    |     # get second point (right) (point2)
    |     # take the center point and move right the radius plus the cushions
    |     p2x = pcx + vecrx * radius + vecrx * cusharound + vecnx * -1 * cushout
    |     p2y = pcy + vecry * radius + vecry * cusharound + vecny * -1 * cushout
    |     p2z = pcz
    | 
    |     # find rxryrz2
    |     # first rotation is 90 degrees about the x- axis
    |     m1 = get_rotation_matrix_from_description("x", -1, 90 * pi / 180)
    |     # second rotation is About 135 degrees about the z+ axis. This calculation is heading1 – 45 degrees
    |     m2 = get_rotation_matrix_from_description("z", 1, heading1 - 45 * pi/180)
    |     # combine them by multiplying
    |     m3 = multiply_matrix(m2, m1)
    |     rxryrz2 = convert_matrix_to_axang(m3)
    |     rx2 = rxryrz2[0]
    |     ry2 = rxryrz2[1]
    |     rz2 = rxryrz2[2]
    | 
    |     point2 = p[p2x, p2y, p2z, rx2, ry2, rz2]
    | 
    |     # get the third point (bottom) (point3)
    |     p3x = pcx + vecnx * -1 * cushout
    |     p3y = pcy + vecny * -1 * cushout
    |     p3z = pcz - vecuz * radius - vecuz * cusharound
    | 
    |     # find rxryrz3
    |     # first rotation is 45 degrees about the y+ axis
    |     m1 = get_rotation_matrix_from_description("y", 1, 45 * pi / 180)
    |     # second rotation is About 180 degrees about the z+ axis. This calculation is heading1 degrees
    |     m2 = get_rotation_matrix_from_description("z", 1, heading1)
    |     # combine them by multiplying
    |     m3 = multiply_matrix(m2, m1)
    |     rxryrz3 = convert_matrix_to_axang(m3)
    |     rx3 = rxryrz3[0]
    |     ry3 = rxryrz3[1]
    |     rz3 = rxryrz3[2]
    | 
    |     point3 = p[p3x, p3y, p3z, rx3, ry3, rz3]
    | 
    |     # get the fourth point (left) (point4)
    |     p4x = pcx - vecrx * radius - vecrx * cusharound + vecnx * -1 * cushout
    |     p4y = pcy - vecry * radius - vecry * cusharound + vecny * -1 * cushout
    |     p4z = pcz
    | 
    |     # find rxryrz4
    |     # first rotation is 90 degrees about the x+ axis
    |     m1 = get_rotation_matrix_from_description("x", 1, 90 * pi / 180)
    |     # second rotation is heading1 + 45 degrees about the z+ axis. approx 225 degrees ccw
    |     m2 = get_rotation_matrix_from_description("z", 1, heading1 + 45 * pi/180)
    |     # combine them by multiplying
    |     m3 = multiply_matrix(m2, m1)
    |     rxryrz4 = convert_matrix_to_axang(m3)
    |     rx4 = rxryrz4[0]
    |     ry4 = rxryrz4[1]
    |     rz4 = rxryrz4[2]
    | 
    |     point4 = p[p4x, p4y, p4z, rx4, ry4, rz4]
    | 
    |     # return the points
    |     ret = struct(point1=point1, point2=point2, point3=point3, point4=point4)
    |     return ret
    | 
    | end
  SuppressedNode
    Script: welder_state_ready()
  SuppressedNode
    sidewallchoice :=  (valueSource=Operator message=Is the sidewall 3/4 inch? valueType=Boolean)
  SuppressedNode
    If sidewallchoice removedSiblings(If(type=Else checkContinuously=false, children(Assignment(valueSource=Expression, variable(name=sidewall), expression=0.375))))
      sidewall := 0.628
  SuppressedNode
    deepcham :=  (valueSource=Operator message=Is the chamfer extra deep? (more than 0.21) valueType=Boolean)
  MoveJ speed 60 deg/s, acceleration 80 deg/s^2 (useActiveTCP=true optimoveEnabled=false optiMoveSpeed=0.3 optiMoveAcceleration=0.09) feature=Base
    Waypoint Waypoint_46: TCP in base x=894.108 y=351.078 z=354.456 mm, rx=2.3264 ry=2.0525 rz=0.0574 rad; joints [-187.182, -67.294, 94.726, 57.522, -0.141, -88.018] deg; TCP offset x=-5.49 y=-328 z=106.39 mm, rx=1.2092 ry=-1.2092 rz=1.2092 rad
  Set NoAction tcp=pretend_w_top
  Script: Test_Teach_Sleeve_Fillet()
  Set NoAction tcp=pretend_w_top
  Script: kill threadId_Thread_1
  Set NoAction tcp=pretend_welder
  SuppressedNode
    path1 := analyze_touchpoints(p11,p12,p21,p22,p3)
  SuppressedNode
    CallSubProgram
  SuppressedNode
    MoveJ speed 60 deg/s, acceleration 80 deg/s^2 (useActiveTCP=true optimoveEnabled=false optiMoveSpeed=0.3 optiMoveAcceleration=0.09) feature=Base
      Waypoint Waypoint_19: TCP in base x=-539.433 y=254.004 z=21.521 mm, rx=-1.7232 ry=0.9213 rz=1.7071 rad; joints [-41.97, -63.602, 146.502, 9.159, 84.533, 189.272] deg; TCP offset x=8.55 y=-271.52 z=102 mm, rx=1.2092 ry=-1.2092 rz=1.2092 rad
  pathturn := main_calculate_sleeve_fillet(tcp_pose_left, tcp_pose_right, tcp_3)
  SuppressedNode
    Folder extrude knife
      lch := get_lift_column_height_condensed()
      If lch > 1
        URCap MachineLogic for Universal Robots (MachineLogic for Universal Robots, Vention Inc.) dataModel(type=addMotor, numberAdded=0, speed_in_mm_per_min=3000.0, acceleration_in_mm_per_s2=50.0, teachColor=BLUE, combo1=MachineMotion1, combo2=(1) Custom Actuator, combo3=Home, combo6=In series, message=Homing, description=Moves the actuator in the negative direction until the home sensor is triggered and sets position to zero (0)., comboAddress=Address 1, comboActuator=Valve 1)
        Script: extrude_knife3()
        URCap MachineLogic for Universal Robots (MachineLogic for Universal Robots, Vention Inc.) dataModel(type=addMotor, numberAdded=0, speed_in_mm_per_min=3000.0, acceleration_in_mm_per_s2=50.0, ActuatorPos=lch, teachColor=BLUE, combo1=MachineMotion1, combo2=(1) Custom Actuator, combo3=Move to Position, combo6=In series, message=Move to Position, description=Moves the actuator to a specified position from the home location., comboAddress=Address 1, comboActuator=Valve 1)
      Else 
        Script: extrude_knife3()
  Script: extrude_knife3()
  SuppressedNode
    Script: move_path_cover_left3()
  SuppressedNode
    pointtopvcham := pathturn[0]
  SuppressedNode
    URCap MachineLogic for Universal Robots (MachineLogic for Universal Robots, Vention Inc.) dataModel(type=addMotor, numberAdded=0, speed_in_mm_per_min=3000.0, acceleration_in_mm_per_s2=50.0, ActuatorPos=liftcolumnzneeded, teachColor=BLUE, combo1=MachineMotion1, combo2=(1) Custom Actuator, combo3=Move to Position, combo6=In series, message=Move to Position, description=Moves the actuator to a specified position from the home location., comboAddress=Address 1, comboActuator=Valve 1)
  SuppressedNode
    MoveJ speed 60 deg/s, acceleration 80 deg/s^2 (useActiveTCP=true optimoveEnabled=false optiMoveSpeed=0.3 optiMoveAcceleration=0.09) feature=Base
      Waypoint Variable (Variable): variable=pointtopvcham
  Script: align_sleeve_fillet_low()
  Script: move_sleeve_fillet_quad()
  MoveJ speed 60 deg/s, acceleration 80 deg/s^2 (useActiveTCP=true optimoveEnabled=false optiMoveSpeed=0.3 optiMoveAcceleration=0.09) feature=Base
    Waypoint Waypoint_8: TCP in base x=-262.599 y=-117.911 z=443.767 mm, rx=0.1153 ry=3.1146 rz=0.2657 rad; joints [5.497, -142.032, 129.309, 13.11, 99.793, -9.621] deg; TCP offset x=-9.5 y=-328 z=105.73 mm, rx=1.2092 ry=-1.2092 rz=1.2092 rad
    Waypoint Waypoint_9: TCP in base x=397.354 y=356.263 z=319.809 mm, rx=2.3163 ry=2.0576 rz=0.0741 rad; joints [-198.308, -118.162, 133.452, -12.561, -11.517, -6.326] deg
  SuppressedNode
    URCap MachineLogic for Universal Robots (MachineLogic for Universal Robots, Vention Inc.) dataModel(type=addMotor, numberAdded=0, speed_in_mm_per_min=3000.0, acceleration_in_mm_per_s2=50.0, teachColor=BLUE, combo1=MachineMotion1, combo2=(1) Custom Actuator, combo3=Home, combo6=In series, message=Homing, description=Moves the actuator in the negative direction until the home sensor is triggered and sets position to zero (0)., comboAddress=Address 1, comboActuator=Valve 1)
  SafeHome (positionOptionType=SPEED_AND_ACCELERATION speed=1.047198 acceleration=1.396263 nextMotionTime=2)
SubProgram Test_Teach_Sleeve_Fillet (keepSynchronizedWithDisk=false) programFile=/programs/Test Teach Sleeve Fillet.urp
  Set NoAction tcp=pretend_w_top
  SuppressedNode
    MoveL speed 250 mm/s, acceleration 1200 mm/s^2 (useActiveTCP=true optimoveEnabled=false optiMoveSpeed=0.3 optiMoveAcceleration=0.09) feature=Base
      Waypoint Waypoint_1: TCP in base x=183.613 y=373.491 z=464.002 mm, rx=0 ry=3.1416 rz=0 rad; joints [-144.817, -120.486, 148.461, -117.931, -90.033, 125.101] deg; TCP offset x=0 y=0 z=19 mm, rx=0 ry=0 rz=0 rad
      'move welder up out of holder'
  MoveJ speed 60 deg/s, acceleration 80 deg/s^2 (useActiveTCP=false optimoveEnabled=false optiMoveSpeed=0.3 optiMoveAcceleration=0.09) tcp=TCP_1_plate; feature=Base
    Waypoint Waypoint_40: TCP in base x=360.688 y=270.12 z=646.145 mm, rx=0.0578 ry=2.126 rz=2.1341 rad; joints [-198.126, -117.852, 133.303, -13.01, -11.422, -6.036] deg
    'above waypoint is home'
    SuppressedNode
      Waypoint Waypoint_2: TCP in base x=-548.957 y=386.285 z=143.71 mm, rx=1.5708 ry=0 rz=0 rad; joints [-60.253, -57.926, 123.544, -65.529, -60.311, -0.099] deg
    SuppressedNode
      Waypoint Waypoint_3: TCP in base x=-565.561 y=-88.282 z=748.934 mm, rx=0.347 ry=3.1015 rz=-0.0385 rad; joints [-12.028, -113.359, 121.362, 263.351, -88.693, -89.284] deg
    Waypoint Waypoint_4: TCP in base x=-946.63 y=32.923 z=107.553 mm, rx=1.1855 ry=-1.4546 rz=-1.2991 rad; joints [-14.723, -32.384, 121.91, 97.274, -87.344, -180.783] deg
  Set NoAction tcp=pretend_w_top
  freedrive_m_var := False
  freedrive_m_var := True
  Popup Message (haltProgram=false message=Move the TCP to point 1 on the edge then click 'Continue' inputType=Text)
  tcp_pose_left := get_actual_tcp_pose()
  freedrive_m_var := False
  Script: sync()
  Wait Sleep waitTime=0.01
  MoveJ speed 60 deg/s, acceleration 80 deg/s^2 (useActiveTCP=true optimoveEnabled=false optiMoveSpeed=0.3 optiMoveAcceleration=0.09) feature=Base
    Waypoint Waypoint_4: TCP in base x=-946.63 y=32.923 z=107.553 mm, rx=1.1855 ry=-1.4546 rz=-1.2991 rad; joints [-14.723, -32.384, 121.91, 97.274, -87.344, -180.783] deg
  MoveJ speed 60 deg/s, acceleration 80 deg/s^2 (useActiveTCP=true optimoveEnabled=false optiMoveSpeed=0.3 optiMoveAcceleration=0.09) feature=Base
    Waypoint Waypoint_5: TCP in base x=-1246.557 y=36.36 z=-286.524 mm, rx=0.3629 ry=-1.2595 rz=-1.7222 rad; joints [1.222, -11.211, 100.501, 238.355, -233.303, -3.079] deg; TCP offset x=-1.032 y=-18.062 z=285.234 mm, rx=0 ry=0 rz=0 rad
  freedrive_m_var := True
  Popup Message (haltProgram=false message=Move the TCP to point 2 on the edge then click 'Continue' inputType=Text)
  tcp_pose_right := get_actual_tcp_pose()
  Popup Message (haltProgram=false message=Move the TCP to point 3 on the edge then click 'Continue' inputType=Text)
  tcp_3 := get_actual_tcp_pose()
  freedrive_m_var := False
  Wait Sleep waitTime=0.25
  Script: sync()
  MoveL speed 100 mm/s, acceleration 1200 mm/s^2 (useActiveTCP=true optimoveEnabled=false optiMoveSpeed=0.3 optiMoveAcceleration=0.09) feature=Base
    MoveDirectionNode expression=[1.0,0.0,-0.5]
      Until DISTANCE (allowActions=false deceleration=3 distanceNodeType=STOP) Distance=0.15; motionParameters(blendRadius=0)
  MoveJ speed 60 deg/s, acceleration 80 deg/s^2 (useActiveTCP=true optimoveEnabled=false optiMoveSpeed=0.3 optiMoveAcceleration=0.09) feature=Base
    Waypoint Waypoint_5: TCP in base x=-1246.557 y=36.36 z=-286.524 mm, rx=0.3629 ry=-1.2595 rz=-1.7222 rad; joints [1.222, -11.211, 100.501, 238.355, -233.303, -3.079] deg
    Waypoint Waypoint_4: TCP in base x=-946.63 y=32.923 z=107.553 mm, rx=1.1855 ry=-1.4546 rz=-1.2991 rad; joints [-14.723, -32.384, 121.91, 97.274, -87.344, -180.783] deg; TCP offset x=0 y=0 z=19 mm, rx=0 ry=0 rz=0 rad
    Waypoint Waypoint_1: TCP in base x=394.188 y=534.376 z=630.191 mm, rx=0.0578 ry=2.126 rz=2.1341 rad; joints [-198.279, -117.801, 133.277, -12.745, -11.485, -6.332] deg; TCP offset x=-1.032 y=-18.062 z=285.234 mm, rx=0 ry=0 rz=0 rad
SubProgram move_sleeve_fillet_quad (keepSynchronizedWithDisk=false) programFile=/programs/move_sleeve_fillet_quad.urp
  Set NoAction tcp=backofhole
  SuppressedNode
    MoveJ speed 60 deg/s, acceleration 80 deg/s^2 (useActiveTCP=true optimoveEnabled=false optiMoveSpeed=0.3 optiMoveAcceleration=0.09) feature=Base
      SuppressedNode
        Waypoint Waypoint_3: TCP in base x=-912.453 y=673.518 z=718.985 mm, rx=-0.4706 ry=-1.9428 rz=0.4955 rad; joints [-63.285, -68.284, 110.161, 88.985, -83.541, -118.353] deg; TCP offset x=-9.5 y=-328 z=105.73 mm, rx=1.2092 ry=-1.2092 rz=1.2092 rad
      SuppressedNode
        Waypoint Waypoint_4: TCP in base x=-1043.534 y=752.126 z=758.241 mm, rx=-0.4498 ry=-2.3257 rz=-0.2665 rad; joints [-53.991, -67.414, 94.218, 102.936, -66.691, -159.337] deg
      Waypoint Waypoint_9: TCP in base x=-850.146 y=808.476 z=769.845 mm, rx=-0.0694 ry=-2.4231 rz=-0.6317 rad; joints [-70.02, -72.001, 93.194, -274.04, -37.901, -142.904] deg
      Waypoint Waypoint_6: TCP in base x=-1042.273 y=808.476 z=769.845 mm, rx=-0.0694 ry=-2.4231 rz=-0.6317 rad; joints [-58.413, -64.349, 84.656, -260.501, -42.539, -159.423] deg
  SuppressedNode
    MoveJ speed 60 deg/s, acceleration 80 deg/s^2 (useActiveTCP=true optimoveEnabled=false optiMoveSpeed=0.3 optiMoveAcceleration=0.09) feature=Base
      SuppressedNode
        Waypoint Waypoint_1: TCP in base x=-1152.594 y=814.679 z=699.964 mm, rx=0.098 ry=-2.3843 rz=-0.4483 rad; joints [-56.525, -54.403, 73.307, 93.455, -42.841, -145.624] deg
      SuppressedNode
        Waypoint Waypoint_5: TCP in base x=-1149.758 y=814.958 z=702.794 mm, rx=-0.0472 ry=-2.3472 rz=-0.7271 rad; joints [-53.278, -57.004, 80.845, -264.711, -44.526, -166.31] deg
      Waypoint Waypoint_7: TCP in base x=-1150.142 y=824.468 z=703.476 mm, rx=-0.1355 ry=-2.1954 rz=-0.513 rad; joints [-54.373, -54.473, 80.141, -274.253, -56.089, -154.835] deg
  SuppressedNode
    MoveP speed 10 mm/s, acceleration 1200 mm/s^2 (blendRadius=0.025 useActiveTCP=true optimoveEnabled=false optiMoveSpeed=0.3 optiMoveAcceleration=0.09) feature=Base
      CircleMove (OrientationMode=FIXED)
        Waypoint ViaPoint_1: TCP in base x=-1137.967 y=888.777 z=671.431 mm, rx=-0.7156 ry=-2.1833 rz=0.6859 rad; joints [-57.632, -55.198, 82.444, 124.608, -82.298, -128.207] deg
        Waypoint EndPoint_1: TCP in base x=-1139.924 y=872.884 z=596.072 mm, rx=-1.219 ry=-0.9297 rz=2.3215 rad; joints [-60.159, -58.197, 98.87, 176.452, -78.393, -68.042] deg
      CircleMove (OrientationMode=FIXED)
        Waypoint ViaPoint_2: TCP in base x=-1155.211 y=763.52 z=646.144 mm, rx=0.9307 ry=-1.6945 rz=-2.1414 rad; joints [-52.747, -75.971, 108.96, 234.472, -18.82, -4.377] deg
        Waypoint Waypoint_1: TCP in base x=-1152.594 y=814.679 z=699.964 mm, rx=0.098 ry=-2.3843 rz=-0.4483 rad; joints [-56.525, -54.403, 73.307, 93.455, -42.841, -145.624] deg
  SuppressedNode
    MoveJ speed 60 deg/s, acceleration 80 deg/s^2 (useActiveTCP=true optimoveEnabled=false optiMoveSpeed=0.3 optiMoveAcceleration=0.09) feature=Base
      SuppressedNode
        Waypoint Waypoint_2: TCP in base x=-917.75 y=830.261 z=524.512 mm, rx=-1.543 ry=-0.8444 rz=1.9881 rad; joints [-66.08, -72.484, 118.808, 175.962, -93.351, -73.55] deg
      Waypoint Waypoint_4: TCP in base x=-1043.534 y=752.126 z=758.241 mm, rx=-0.4498 ry=-2.3257 rz=-0.2665 rad; joints [-53.991, -67.414, 94.218, 102.936, -66.691, -159.337] deg
      Waypoint Waypoint_8: TCP in base x=-754.583 y=757.082 z=772.781 mm, rx=-0.4498 ry=-2.3257 rz=-0.2665 rad; joints [-73.782, -79.343, 107.572, 92.439, -55.198, -140.846] deg
  SuppressedNode
    Folder half circle
      MoveJ speed 60 deg/s, acceleration 80 deg/s^2 (useActiveTCP=true optimoveEnabled=false optiMoveSpeed=0.3 optiMoveAcceleration=0.09) feature=Base
        Waypoint Waypoint_13: TCP in base x=-1410.884 y=263.861 z=-13.194 mm, rx=-0.2057 ry=-2.2742 rz=-0.4378 rad; joints [-18.611, -21.126, 85.064, -293.08, -78.09, -188.172] deg
      MoveJ speed 60 deg/s, acceleration 80 deg/s^2 (useActiveTCP=true optimoveEnabled=false optiMoveSpeed=0.3 optiMoveAcceleration=0.09) feature=Base
        Waypoint Waypoint_10: TCP in base x=-1440.647 y=263.861 z=-48.062 mm, rx=-0.2057 ry=-2.2742 rz=-0.4378 rad; joints [-18.086, -18.126, 80.761, -291.695, -78.433, -188.577] deg
        SuppressedNode
          Waypoint Waypoint_11: TCP in base x=-1286.175 y=549.195 z=115.468 mm, rx=-0.27 ry=-1.5277 rz=-1.42 rad; joints [-20.499, -22.138, 88.563, -259.74, -128.557, -138.212] deg; TCP offset x=-1.032 y=-18.062 z=285.234 mm, rx=0 ry=0 rz=0 rad
        SuppressedNode
          Waypoint Waypoint_12: TCP in base x=-1198.19 y=495.746 z=-342.486 mm, rx=-1.4417 ry=-1.7142 rz=-0.5215 rad; joints [-20.358, -19.189, 100.698, -215.464, -126.338, -45.331] deg
      MoveP speed 8 mm/s, acceleration 1200 mm/s^2 (blendRadius=0.025 useActiveTCP=true optimoveEnabled=false optiMoveSpeed=0.3 optiMoveAcceleration=0.09) feature=Base
        CircleMove (OrientationMode=FIXED)
          Waypoint ViaPoint_3: TCP in base x=-1436.982 y=288.423 z=-164.849 mm, rx=-1.2985 ry=-1.3493 rz=1.8084 rad; joints [-22.4, -18.108, 96.782, -229.781, -128.579, -68.735] deg; TCP offset x=-9.5 y=-328 z=105.73 mm, rx=1.2092 ry=-1.2092 rz=1.2092 rad
          Waypoint EndPoint_2: TCP in base x=-1450.471 y=225.502 z=-193.907 mm, rx=-1.3296 ry=-0.3697 rz=2.6077 rad; joints [-22.267, -13.945, 97.987, -213.988, -92.35, -25.678] deg
      MoveJ speed 60 deg/s, acceleration 80 deg/s^2 (useActiveTCP=true optimoveEnabled=false optiMoveSpeed=0.3 optiMoveAcceleration=0.09) feature=Base
        Waypoint Waypoint_14: TCP in base x=-1380.88 y=218.821 z=-252.804 mm, rx=-1.3435 ry=-0.3935 rz=2.6113 rad; joints [-23.838, -10.524, 100.952, -220.078, -91.217, -28.02] deg
  Folder assign points
    p1 := pathturn[0]
    p2 := pathturn[1]
    p3 := pathturn[2]
    p4 := pathturn[3]
    pa1 := p[p1[0]+0.05,p1[1],p1[2]+0.05,p1[3],p1[4],p1[5]]
  Folder full circle
    SuppressedNode
      MoveJ speed 60 deg/s, acceleration 80 deg/s^2 (useActiveTCP=true optimoveEnabled=false optiMoveSpeed=0.3 optiMoveAcceleration=0.09) feature=Base
        'start point example'
        Waypoint Waypoint_13: TCP in base x=-1410.884 y=263.861 z=-13.194 mm, rx=-0.2057 ry=-2.2742 rz=-0.4378 rad; joints [-18.611, -21.126, 85.064, -293.08, -78.09, -188.172] deg
    MoveJ speed 60 deg/s, acceleration 80 deg/s^2 (useActiveTCP=true optimoveEnabled=false optiMoveSpeed=0.3 optiMoveAcceleration=0.09) feature=Base
      SuppressedNode
        Waypoint Waypoint_10: TCP in base x=-1440.647 y=263.861 z=-48.062 mm, rx=-0.2057 ry=-2.2742 rz=-0.4378 rad; joints [-18.086, -18.126, 80.761, -291.695, -78.433, -188.577] deg
      SuppressedNode
        Waypoint Waypoint_11: TCP in base x=-1286.175 y=549.195 z=115.468 mm, rx=-0.27 ry=-1.5277 rz=-1.42 rad; joints [-20.499, -22.138, 88.563, -259.74, -128.557, -138.212] deg; TCP offset x=-1.032 y=-18.062 z=285.234 mm, rx=0 ry=0 rz=0 rad
      SuppressedNode
        Waypoint Waypoint_12: TCP in base x=-1198.19 y=495.746 z=-342.486 mm, rx=-1.4417 ry=-1.7142 rz=-0.5215 rad; joints [-20.358, -19.189, 100.698, -215.464, -126.338, -45.331] deg
      Waypoint Variable (Variable): variable=pa1
      Waypoint Variable (Variable): variable=p1
    SuppressedNode
      MoveP speed 8 mm/s, acceleration 1200 mm/s^2 (blendRadius=0.025 useActiveTCP=true optimoveEnabled=false optiMoveSpeed=0.3 optiMoveAcceleration=0.09) feature=Base
        CircleMove (OrientationMode=FIXED)
          Waypoint ViaPoint_3: TCP in base x=-1436.982 y=288.423 z=-164.849 mm, rx=-1.2985 ry=-1.3493 rz=1.8084 rad; joints [-22.4, -18.108, 96.782, -229.781, -128.579, -68.735] deg; TCP offset x=-9.5 y=-328 z=105.73 mm, rx=1.2092 ry=-1.2092 rz=1.2092 rad
          Waypoint EndPoint_2: TCP in base x=-1450.471 y=225.502 z=-193.907 mm, rx=-1.3296 ry=-0.3697 rz=2.6077 rad; joints [-22.267, -13.945, 97.987, -213.988, -92.35, -25.678] deg
        CircleMove (OrientationMode=FIXED)
          Waypoint ViaPoint_4: TCP in base x=-1458.06 y=174.729 z=-155.961 mm, rx=0.9854 ry=-0.8297 rz=-2.4175 rad; joints [-21.89, -10.796, 94.59, -213.949, -40.159, 6.455] deg
          Waypoint EndPoint_3: TCP in base x=-1453.174 y=244.554 z=-53.456 mm, rx=-0.0081 ry=-2.2253 rz=-0.4366 rad; joints [-20.236, -35.116, 108.931, -127.571, 69.187, -2.082] deg
    MoveP speed 10 mm/s, acceleration 1200 mm/s^2 (blendRadius=0.025 useActiveTCP=true optimoveEnabled=false optiMoveSpeed=0.3 optiMoveAcceleration=0.09) feature=Base
      CircleMove (OrientationMode=FIXED)
        Waypoint Variable (Variable): variable=p2
        Waypoint Variable (Variable): variable=p3
      CircleMove (OrientationMode=FIXED)
        Waypoint Variable (Variable): variable=p4
        Waypoint Variable (Variable): variable=p1
    MoveL speed 250 mm/s, acceleration 1200 mm/s^2 (useActiveTCP=true optimoveEnabled=false optiMoveSpeed=0.3 optiMoveAcceleration=0.09) feature=Base
      MoveDirectionNode expression=[1.0,0.0,1.0]
        Until DISTANCE (allowActions=false deceleration=3 distanceNodeType=STOP) Distance=0.1; motionParameters(blendRadius=0)
    Popup Message (haltProgram=true message=pause inputType=Text)
    MoveJ speed 60 deg/s, acceleration 80 deg/s^2 (useActiveTCP=true optimoveEnabled=false optiMoveSpeed=0.3 optiMoveAcceleration=0.09) feature=Base
      Waypoint Waypoint_3: TCP in base x=-1407.381 y=244.554 z=7.478 mm, rx=-0.0081 ry=-2.2253 rz=-0.4366 rad; joints [-21.148, -40.183, 113.996, -127.853, 68.651, -1.292] deg
      Waypoint Waypoint_6: TCP in base x=-1318.966 y=244.554 z=7.478 mm, rx=1.059 ry=-2.1109 rz=-0.921 rad; joints [-32.341, -42.763, 117.442, -171.905, 11.465, 43.721] deg
  SuppressedNode
    MoveJ speed 60 deg/s, acceleration 80 deg/s^2 (useActiveTCP=true optimoveEnabled=false optiMoveSpeed=0.3 optiMoveAcceleration=0.09) feature=Base
      'oldhome'
      Waypoint Waypoint_17: TCP in base x=397.38 y=356.254 z=319.821 mm, rx=2.3163 ry=2.0576 rz=0.0741 rad; joints [-198.308, -118.162, 133.451, -12.562, -11.515, -6.325] deg
  SuppressedNode
    MoveJ speed 60 deg/s, acceleration 80 deg/s^2 (useActiveTCP=true optimoveEnabled=false optiMoveSpeed=0.3 optiMoveAcceleration=0.09) feature=Base
      Waypoint Waypoint_18: TCP in base x=-108.326 y=728.695 z=730.15 mm, rx=-0.9793 ry=0.0055 rz=2.4246 rad; joints [-134.638, -102.677, 135.598, -114.689, -40.923, -114.839] deg
  SuppressedNode
    MoveJ speed 60 deg/s, acceleration 80 deg/s^2 (useActiveTCP=true optimoveEnabled=false optiMoveSpeed=0.3 optiMoveAcceleration=0.09) feature=Base
      Waypoint Waypoint_19: TCP in base x=-1040.406 y=263.861 z=-13.194 mm, rx=-0.2057 ry=-2.2742 rz=-0.4378 rad; joints [-29.173, -26.842, 118.297, -322.804, -71.321, -179.763] deg
  SuppressedNode
    MoveJ speed 60 deg/s, acceleration 80 deg/s^2 (useActiveTCP=true optimoveEnabled=false optiMoveSpeed=0.3 optiMoveAcceleration=0.09) feature=Base
      'example start'
      Waypoint Waypoint_13: TCP in base x=-1410.884 y=263.861 z=-13.194 mm, rx=-0.2057 ry=-2.2742 rz=-0.4378 rad; joints [-18.611, -21.126, 85.064, -293.08, -78.09, -188.172] deg
SubProgram move_path_cover_lt (keepSynchronizedWithDisk=false) programFile=/programs/move_path_cover_lt.urp
  p1 := pathturn[1]
  p2 := pathturn[2]
  p3 := pathturn[3]
  p4 := pathturn[4]
  p5 := pathturn[5]
  p6 := pathturn[6]
  pa1 := p[p1[0],p1[1],p1[2]+0.05,p1[3],p1[4],p1[5]]
  pret := p[p6[0],p6[1],p6[2]+0.05,p6[3],p6[4],p6[5]]
  'go to preheat'
  Set NoAction tcp=pretend_welder
  MoveJ speed 60 deg/s, acceleration 80 deg/s^2 (useActiveTCP=true optimoveEnabled=false optiMoveSpeed=0.3 optiMoveAcceleration=0.09) feature=Base
    Waypoint Variable (Variable): variable=pa1
  MoveL speed 50 mm/s, acceleration 50 mm/s^2 (useActiveTCP=true optimoveEnabled=false optiMoveSpeed=0.3 optiMoveAcceleration=0.09) feature=Base
    Waypoint Variable (Variable): variable=p1
  Wait Sleep waitTime=4
  URCap WireTank Serial (WireTank Serial, WireTank, LLC) dataModel(NODE_TITLE=Serial Bridge uR1, Command=[252,82,49], QUERY=false, byte_array=true, OUTPUT_ENTRY=Static, Variable(key=OUTPUT_VARIABLE, variable(name=HwResp)))
  Set DigitalOutput pin=digital_out[0]; digitalValue=1
  Wait Sleep waitTime=1
  MoveL speed 9 mm/s, acceleration 1200 mm/s^2 (useActiveTCP=true optimoveEnabled=false optiMoveSpeed=0.3 optiMoveAcceleration=0.09) feature=Base
    Waypoint Variable (Variable): variable=p2
    Waypoint Variable (Variable): variable=p3
    Waypoint Variable (Variable): variable=p4
    Waypoint Variable (Variable): variable=p5
  SuppressedNode
    If deepcham removedSiblings(If(type=Else checkContinuously=false, children(Move(motionType=MoveL speed=0.01 acceleration=1.2 useActiveTCP=true positionType=CartesianPose optimoveEnabled=false optiMoveSpeed=0.3 optiMoveAcceleration=0.09, feature=Base, children(Waypoint(type=Variable name=Variable, variable=p2), Waypoint(type=Variable name=Variable, variable=p3), Waypoint(type=Variable name=Variable, variable=p4), Waypoint(type=Variable name=Variable, variable=p5))))))
      MoveL speed 7 mm/s, acceleration 1200 mm/s^2 (useActiveTCP=true optimoveEnabled=false optiMoveSpeed=0.3 optiMoveAcceleration=0.09) feature=Base
        Waypoint Variable (Variable): variable=p2
        Waypoint Variable (Variable): variable=p3
        Waypoint Variable (Variable): variable=p4
        Waypoint Variable (Variable): variable=p5
  URCap WireTank Serial (WireTank Serial, WireTank, LLC) dataModel(QUERY=false, byte_array=true, NODE_TITLE=Serial Bridge uR0, Command=[252,82,48], OUTPUT_ENTRY=Static, Variable(key=OUTPUT_VARIABLE, variable(name=HwResp)))
  Set DigitalOutput pin=digital_out[0]; digitalValue=0
  MoveL speed 10 mm/s, acceleration 1200 mm/s^2 (useActiveTCP=true optimoveEnabled=false optiMoveSpeed=0.3 optiMoveAcceleration=0.09) feature=Base
    Waypoint Variable (Variable): variable=p6
  Wait Sleep waitTime=1
  MoveL speed 50 mm/s, acceleration 50 mm/s^2 (useActiveTCP=true optimoveEnabled=false optiMoveSpeed=0.3 optiMoveAcceleration=0.09) feature=Base
    Waypoint Variable (Variable): variable=pret
SubProgram align_sleeve_fillet_low (keepSynchronizedWithDisk=false) programFile=/programs/align_sleeve_fillet_low.urp
  Set NoAction tcp=pretend_welder
  SuppressedNode
    MoveJ speed 60 deg/s, acceleration 80 deg/s^2 (useActiveTCP=true optimoveEnabled=false optiMoveSpeed=0.3 optiMoveAcceleration=0.09) feature=Base
      SuppressedNode
        Waypoint Waypoint_3: TCP in base x=-912.453 y=673.518 z=718.985 mm, rx=-0.4706 ry=-1.9428 rz=0.4955 rad; joints [-63.285, -68.284, 110.161, 88.985, -83.541, -118.353] deg
      SuppressedNode
        Waypoint Waypoint_4: TCP in base x=-1043.534 y=752.126 z=758.241 mm, rx=-0.4498 ry=-2.3257 rz=-0.2665 rad; joints [-53.991, -67.414, 94.218, 102.936, -66.691, -159.337] deg
      Waypoint Waypoint_9: TCP in base x=-850.146 y=808.476 z=769.845 mm, rx=-0.0694 ry=-2.4231 rz=-0.6317 rad; joints [-70.02, -72.001, 93.194, -274.04, -37.901, -142.904] deg
      Waypoint Waypoint_6: TCP in base x=-1042.273 y=808.476 z=769.845 mm, rx=-0.0694 ry=-2.4231 rz=-0.6317 rad; joints [-58.413, -64.349, 84.656, -260.501, -42.539, -159.423] deg
  SuppressedNode
    MoveJ speed 60 deg/s, acceleration 80 deg/s^2 (useActiveTCP=true optimoveEnabled=false optiMoveSpeed=0.3 optiMoveAcceleration=0.09) feature=Base
      SuppressedNode
        Waypoint Waypoint_1: TCP in base x=-1152.594 y=814.679 z=699.964 mm, rx=0.098 ry=-2.3843 rz=-0.4483 rad; joints [-56.525, -54.403, 73.307, 93.455, -42.841, -145.624] deg
      SuppressedNode
        Waypoint Waypoint_5: TCP in base x=-1149.758 y=814.958 z=702.794 mm, rx=-0.0472 ry=-2.3472 rz=-0.7271 rad; joints [-53.278, -57.004, 80.845, -264.711, -44.526, -166.31] deg
      Waypoint Waypoint_7: TCP in base x=-1150.142 y=824.468 z=703.476 mm, rx=-0.1355 ry=-2.1954 rz=-0.513 rad; joints [-54.373, -54.473, 80.141, -274.253, -56.089, -154.835] deg
  SuppressedNode
    MoveP speed 10 mm/s, acceleration 1200 mm/s^2 (blendRadius=0.025 useActiveTCP=true optimoveEnabled=false optiMoveSpeed=0.3 optiMoveAcceleration=0.09) feature=Base
      CircleMove (OrientationMode=FIXED)
        Waypoint ViaPoint_1: TCP in base x=-1137.967 y=888.777 z=671.431 mm, rx=-0.7156 ry=-2.1833 rz=0.6859 rad; joints [-57.632, -55.198, 82.444, 124.608, -82.298, -128.207] deg
        Waypoint EndPoint_1: TCP in base x=-1139.924 y=872.884 z=596.072 mm, rx=-1.219 ry=-0.9297 rz=2.3215 rad; joints [-60.159, -58.197, 98.87, 176.452, -78.393, -68.042] deg
      CircleMove (OrientationMode=FIXED)
        Waypoint ViaPoint_2: TCP in base x=-1155.211 y=763.52 z=646.144 mm, rx=0.9307 ry=-1.6945 rz=-2.1414 rad; joints [-52.747, -75.971, 108.96, 234.472, -18.82, -4.377] deg
        Waypoint Waypoint_1: TCP in base x=-1152.594 y=814.679 z=699.964 mm, rx=0.098 ry=-2.3843 rz=-0.4483 rad; joints [-56.525, -54.403, 73.307, 93.455, -42.841, -145.624] deg
  SuppressedNode
    MoveJ speed 60 deg/s, acceleration 80 deg/s^2 (useActiveTCP=true optimoveEnabled=false optiMoveSpeed=0.3 optiMoveAcceleration=0.09) feature=Base
      SuppressedNode
        Waypoint Waypoint_2: TCP in base x=-917.75 y=830.261 z=524.512 mm, rx=-1.543 ry=-0.8444 rz=1.9881 rad; joints [-66.08, -72.484, 118.808, 175.962, -93.351, -73.55] deg
      Waypoint Waypoint_4: TCP in base x=-1043.534 y=752.126 z=758.241 mm, rx=-0.4498 ry=-2.3257 rz=-0.2665 rad; joints [-53.991, -67.414, 94.218, 102.936, -66.691, -159.337] deg
      Waypoint Waypoint_8: TCP in base x=-754.583 y=757.082 z=772.781 mm, rx=-0.4498 ry=-2.3257 rz=-0.2665 rad; joints [-73.782, -79.343, 107.572, 92.439, -55.198, -140.846] deg
  SuppressedNode
    Folder half circle
      MoveJ speed 60 deg/s, acceleration 80 deg/s^2 (useActiveTCP=true optimoveEnabled=false optiMoveSpeed=0.3 optiMoveAcceleration=0.09) feature=Base
        Waypoint Waypoint_13: TCP in base x=-1410.884 y=263.861 z=-13.194 mm, rx=-0.2057 ry=-2.2742 rz=-0.4378 rad; joints [-18.611, -21.126, 85.064, -293.08, -78.09, -188.172] deg
      MoveJ speed 60 deg/s, acceleration 80 deg/s^2 (useActiveTCP=true optimoveEnabled=false optiMoveSpeed=0.3 optiMoveAcceleration=0.09) feature=Base
        Waypoint Waypoint_10: TCP in base x=-1440.647 y=263.861 z=-48.062 mm, rx=-0.2057 ry=-2.2742 rz=-0.4378 rad; joints [-18.086, -18.126, 80.761, -291.695, -78.433, -188.577] deg
        SuppressedNode
          Waypoint Waypoint_11: TCP in base x=-1286.175 y=549.195 z=115.468 mm, rx=-0.27 ry=-1.5277 rz=-1.42 rad; joints [-20.499, -22.138, 88.563, -259.74, -128.557, -138.212] deg; TCP offset x=-1.032 y=-18.062 z=285.234 mm, rx=0 ry=0 rz=0 rad
        SuppressedNode
          Waypoint Waypoint_12: TCP in base x=-1198.19 y=495.746 z=-342.486 mm, rx=-1.4417 ry=-1.7142 rz=-0.5215 rad; joints [-20.358, -19.189, 100.698, -215.464, -126.338, -45.331] deg
      MoveP speed 8 mm/s, acceleration 1200 mm/s^2 (blendRadius=0.025 useActiveTCP=true optimoveEnabled=false optiMoveSpeed=0.3 optiMoveAcceleration=0.09) feature=Base
        CircleMove (OrientationMode=FIXED)
          Waypoint ViaPoint_3: TCP in base x=-1436.982 y=288.423 z=-164.849 mm, rx=-1.2985 ry=-1.3493 rz=1.8084 rad; joints [-22.4, -18.108, 96.782, -229.781, -128.579, -68.735] deg; TCP offset x=-9.5 y=-328 z=105.73 mm, rx=1.2092 ry=-1.2092 rz=1.2092 rad
          Waypoint EndPoint_2: TCP in base x=-1450.471 y=225.502 z=-193.907 mm, rx=-1.3296 ry=-0.3697 rz=2.6077 rad; joints [-22.267, -13.945, 97.987, -213.988, -92.35, -25.678] deg
      MoveJ speed 60 deg/s, acceleration 80 deg/s^2 (useActiveTCP=true optimoveEnabled=false optiMoveSpeed=0.3 optiMoveAcceleration=0.09) feature=Base
        Waypoint Waypoint_14: TCP in base x=-1380.88 y=218.821 z=-252.804 mm, rx=-1.3435 ry=-0.3935 rz=2.6113 rad; joints [-23.838, -10.524, 100.952, -220.078, -91.217, -28.02] deg
  SuppressedNode
    Folder full circle
      MoveJ speed 60 deg/s, acceleration 80 deg/s^2 (useActiveTCP=true optimoveEnabled=false optiMoveSpeed=0.3 optiMoveAcceleration=0.09) feature=Base
        'start point example'
        Waypoint Waypoint_13: TCP in base x=-1410.884 y=263.861 z=-13.194 mm, rx=-0.2057 ry=-2.2742 rz=-0.4378 rad; joints [-18.611, -21.126, 85.064, -293.08, -78.09, -188.172] deg
      MoveJ speed 60 deg/s, acceleration 80 deg/s^2 (useActiveTCP=true optimoveEnabled=false optiMoveSpeed=0.3 optiMoveAcceleration=0.09) feature=Base
        Waypoint Waypoint_10: TCP in base x=-1440.647 y=263.861 z=-48.062 mm, rx=-0.2057 ry=-2.2742 rz=-0.4378 rad; joints [-18.086, -18.126, 80.761, -291.695, -78.433, -188.577] deg
        SuppressedNode
          Waypoint Waypoint_11: TCP in base x=-1286.175 y=549.195 z=115.468 mm, rx=-0.27 ry=-1.5277 rz=-1.42 rad; joints [-20.499, -22.138, 88.563, -259.74, -128.557, -138.212] deg; TCP offset x=-1.032 y=-18.062 z=285.234 mm, rx=0 ry=0 rz=0 rad
        SuppressedNode
          Waypoint Waypoint_12: TCP in base x=-1198.19 y=495.746 z=-342.486 mm, rx=-1.4417 ry=-1.7142 rz=-0.5215 rad; joints [-20.358, -19.189, 100.698, -215.464, -126.338, -45.331] deg
      MoveP speed 8 mm/s, acceleration 1200 mm/s^2 (blendRadius=0.025 useActiveTCP=true optimoveEnabled=false optiMoveSpeed=0.3 optiMoveAcceleration=0.09) feature=Base
        CircleMove (OrientationMode=FIXED)
          Waypoint ViaPoint_3: TCP in base x=-1436.982 y=288.423 z=-164.849 mm, rx=-1.2985 ry=-1.3493 rz=1.8084 rad; joints [-22.4, -18.108, 96.782, -229.781, -128.579, -68.735] deg; TCP offset x=-9.5 y=-328 z=105.73 mm, rx=1.2092 ry=-1.2092 rz=1.2092 rad
          Waypoint EndPoint_2: TCP in base x=-1450.471 y=225.502 z=-193.907 mm, rx=-1.3296 ry=-0.3697 rz=2.6077 rad; joints [-22.267, -13.945, 97.987, -213.988, -92.35, -25.678] deg
        CircleMove (OrientationMode=FIXED)
          Waypoint ViaPoint_4: TCP in base x=-1458.06 y=174.729 z=-155.961 mm, rx=0.9854 ry=-0.8297 rz=-2.4175 rad; joints [-21.89, -10.796, 94.59, -213.949, -40.159, 6.455] deg
          Waypoint EndPoint_3: TCP in base x=-1453.174 y=244.554 z=-53.456 mm, rx=-0.0081 ry=-2.2253 rz=-0.4366 rad; joints [-20.236, -35.116, 108.931, -127.571, 69.187, -2.082] deg
      MoveL speed 250 mm/s, acceleration 1200 mm/s^2 (useActiveTCP=true optimoveEnabled=false optiMoveSpeed=0.3 optiMoveAcceleration=0.09) feature=Base
        MoveDirectionNode expression=[1.0,0.0,1.0]
          Until DISTANCE (allowActions=false deceleration=3 distanceNodeType=STOP) Distance=0.1; motionParameters(blendRadius=0)
      MoveJ speed 60 deg/s, acceleration 80 deg/s^2 (useActiveTCP=true optimoveEnabled=false optiMoveSpeed=0.3 optiMoveAcceleration=0.09) feature=Base
        Waypoint Waypoint_15: TCP in base x=-1407.381 y=244.554 z=7.478 mm, rx=-0.0081 ry=-2.2253 rz=-0.4366 rad; joints [-21.148, -40.183, 113.996, -127.853, 68.651, -1.292] deg
        Waypoint Waypoint_16: TCP in base x=-1318.966 y=244.554 z=7.478 mm, rx=1.059 ry=-2.1109 rz=-0.921 rad; joints [-32.341, -42.763, 117.442, -171.905, 11.465, 43.721] deg
  MoveJ speed 60 deg/s, acceleration 80 deg/s^2 (useActiveTCP=true optimoveEnabled=false optiMoveSpeed=0.3 optiMoveAcceleration=0.09) feature=Base
    'oldhome'
    Waypoint Waypoint_17: TCP in base x=397.38 y=356.254 z=319.821 mm, rx=2.3163 ry=2.0576 rz=0.0741 rad; joints [-198.308, -118.162, 133.451, -12.562, -11.515, -6.325] deg
  MoveJ speed 60 deg/s, acceleration 80 deg/s^2 (useActiveTCP=true optimoveEnabled=false optiMoveSpeed=0.3 optiMoveAcceleration=0.09) feature=Base
    Waypoint Waypoint_18: TCP in base x=-108.326 y=728.695 z=730.15 mm, rx=-0.9793 ry=0.0055 rz=2.4246 rad; joints [-134.638, -102.677, 135.598, -114.689, -40.923, -114.839] deg
  MoveJ speed 60 deg/s, acceleration 80 deg/s^2 (useActiveTCP=true optimoveEnabled=false optiMoveSpeed=0.3 optiMoveAcceleration=0.09) feature=Base
    Waypoint Waypoint_2: TCP in base x=-1040.406 y=263.861 z=-13.194 mm, rx=-0.2057 ry=-2.2742 rz=-0.4378 rad; joints [-29.173, -26.842, 118.297, -322.804, -71.321, -179.763] deg
  SuppressedNode
    MoveJ speed 60 deg/s, acceleration 80 deg/s^2 (useActiveTCP=true optimoveEnabled=false optiMoveSpeed=0.3 optiMoveAcceleration=0.09) feature=Base
      'example start'
      Waypoint Waypoint_13: TCP in base x=-1410.884 y=263.861 z=-13.194 mm, rx=-0.2057 ry=-2.2742 rz=-0.4378 rad; joints [-18.611, -21.126, 85.064, -293.08, -78.09, -188.172] deg
SubProgram extrude_knife3 (keepSynchronizedWithDisk=false) programFile=/programs/extrude_knife3.urp
  Folder pre program stuff
    Set NoAction tcp=pretend_welder
    ek_sp := get_actual_tcp_pose()
    MoveL speed 5 mm/s, acceleration 1200 mm/s^2 (useActiveTCP=true optimoveEnabled=false optiMoveSpeed=0.3 optiMoveAcceleration=0.09) feature=Base
      Waypoint Variable (Variable): variable=ek_sp
    SuppressedNode
      Script file /programs/analyze_touchpoints.script
        | # this file creates the function for analyzing touchpoints
        | # define pi
        | pi = 3.1415926535
        | # initialize a lift column extension needed of 0.0
        | global liftcolumnzneeded = 0.0
        | 
        | # this is the main entry point for calculations.
        | # it takes in the 5 points, analyzes the shape of the box, and then calculates path points and returns them
        | # specifically for Down, Over, then Around (DOtA)
        | # specifically for right-sided boxes (vertical weld on right side of edge)
        | def main_calculate_right(p11, p12, p21, p22, p3, p13, p23, chamferover):
        |     struct1 = analyze_touchpoints_only(p11, p12, p21, p22, p3)
        |     list1 = analyze_vertical_touchpoints(p11, p12, p13, p21, p22, p23, p3)
        |     struct2 = calculate_DOtA_points_right(struct1, list1, chamferover)
        |     validity = check_validity_right(struct1, struct2)
        |     return struct2
        | end
        | 
        | # this is the main entry point for calculations.
        | # it takes in the 5 points, analyzes the shape of the box, and then calculates path points and returns them
        | # specifically for Down, Over, then Around (DOtA)
        | # specifically for left-sided boxes (vertical weld on left side of edge)
        | def main_calculate_left(p11, p12, p21, p22, p3, p13, p23, chamferover):
        |     struct1 = analyze_touchpoints_only(p11, p12, p21, p22, p3)
        |     list1 = analyze_vertical_touchpoints(p11, p12, p13, p21, p22, p23, p3)
        |     struct2 = calculate_DOtA_points_left(struct1, list1, chamferover)
        |     validity = check_validity_left(struct1, struct2)
        |     return struct2
        | end
        | 
        | # this is the main entry point for calculations, for Floor Corner Extended.
        | # it takes in the 7 touchpoints, analyzes the shape of the box.
        | # takes in the user defined point for the top of the weld (tcp_pose_top) and then calculates path points
        | # loopingly tries to calculate the extension along the sidewall that fulfills get_inverse_kin_has_solution() and provides the farthest extension possible
        | # returns the pathpoints
        | # specifically for Down, Over, then Around (DOtA)
        | # specifically for right-sided boxes (vertical weld on right side of edge)
        | def main_calculate_right_extended(p11, p12, p21, p22, p3, p13, p23, chamferover, chamferup, tcp_pose_top):
        |     struct1 = analyze_touchpoints_only(p11, p12, p21, p22, p3)
        |     list1 = analyze_vertical_touchpoints(p11, p12, p13, p21, p22, p23, p3)
        |     struct2 = calculate_DOtA_points_right_extended(struct1, list1, chamferover, chamferup, tcp_pose_top)
        |     struct3 = check_validity_right(struct1, struct2)
        |     return struct3
        | end
        | 
        | # this is the main entry point for calculations, for Floor Corner Extended.
        | # it takes in the 7 touchpoints, analyzes the shape of the box.
        | # takes in the user defined point for the top of the weld (tcp_pose_top) and then calculates path points
        | # loopingly tries to calculate the extension along the sidewall that fulfills get_inverse_kin_has_solution() and provides the farthest extension possible
        | # returns the pathpoints
        | # specifically for Down, Over, then Around (DOtA)
        | # specifically for left-sided boxes (vertical weld on left side of edge)
        | def main_calculate_left_extended(p11, p12, p21, p22, p3, p13, p23, chamferover, chamferup, tcp_pose_top):
        |     struct1 = analyze_touchpoints_only(p11, p12, p21, p22, p3)
        |     list1 = analyze_vertical_touchpoints(p11, p12, p13, p21, p22, p23, p3)
        |     struct2 = calculate_DOtA_points_left_extended(struct1, list1, chamferover, chamferup, tcp_pose_top)
        |     struct3 = check_validity_left(struct1, struct2)
        |     return struct3
        | end
        | 
        | # it takes 5 arguments as points
        | # it returns a struct containing: (pointintersect, pointapproach1, pointapproach2, point1, point2, point3, point4, point5, pointreturn1, heading1, heading2, heading3, path2r1, path2r2, path2l1, path2l2)
        | # specifically for Around then Up (AtU)
        | def analyze_touchpoints(p11, p12, p21, p22, p3):
        |   # FIND THE INTERSECTION
        |   # comment get the z
        |   zcoord=p3[2]
        | 
        |   # get the raw points from the first line
        |   l1p1x=p11[0]
        |   l1p1y=p11[1]
        |   l1p2x=p12[0]
        |   l1p2y=p12[1]
        | 
        |   # equate the first line in 2d space
        |   ml1 = (l1p2y-l1p1y) / (l1p2x-l1p1x)
        | 
        |   # b = y - mx
        |   bl1 = l1p1y - ml1 * l1p1x
        | 
        |   # get the raw points from the second line
        |   l2p1x=p21[0]
        |   l2p1y=p21[1]
        |   l2p2x=p22[0]
        |   l2p2y=p22[1]
        | 
        |   # equate the second line in 2d space
        |   ml2 = (l2p2y-l2p1y) / (l2p2x-l2p1x)
        | 
        |   # b = y - mx
        |   bl2 = l2p1y - ml2 * l2p1x
        | 
        | 
        |   # find the intersection of the two lines
        |   # m1x+b1 = m2x+b2
        |   # m1x - m2x = b2 - b1
        |   # x = (b2-b1) / (m1-m2)
        |   xintersect = (bl2-bl1) / (ml1-ml2)
        |   yintersect = ml1 * xintersect + bl1
        | 
        |   #FIND THE VECTORS
        |   #define a vector from the intersection to the second point on the first line
        |   l1delxfull = l1p2x - xintersect
        |   l1delyfull = l1p2y - yintersect
        | 
        |   l1delmag = sqrt(l1delxfull*l1delxfull + l1delyfull*l1delyfull)
        | 
        |   l1delxunit = l1delxfull / l1delmag
        |   l1delyunit = l1delyfull / l1delmag
        | 
        |   #define a vector from the intersection to the second point on the second line
        |   l2delxfull = l2p2x - xintersect
        |   l2delyfull = l2p2y - yintersect
        | 
        |   l2delmag = sqrt(l2delxfull*l2delxfull + l2delyfull*l2delyfull)
        | 
        |   l2delxunit = l2delxfull / l2delmag
        |   l2delyunit = l2delyfull / l2delmag
        | 
        |   # FIND THE FOUR POINTS ON THE LINES
        |   # find locations 8 inches away from  intersect point
        |   # CONST
        |   welddistance = 8
        |   roundoverdistance = 0.05
        |   zup = .375
        |   # inches
        |   wd = welddistance * 25.4 / 1000
        |   rod = roundoverdistance * 25.4 / 1000
        |   zup = zup * 25.4 / 1000
        | 
        |   # now we have the unit vector. extend the weld distance from the intersection
        |   x = xintersect + l1delxunit * wd
        |   y = yintersect + l1delyunit * wd
        |   z = zcoord + zup
        | 
        |   point1 = p[x,y,z,1.570796,0,0] # dummy orientation for now
        | 
        |   x = xintersect + l1delxunit * rod
        |   y = yintersect + l1delyunit * rod
        | 
        |   point2 = p[x,y,z,1.570796,0,0]
        | 
        |   # now we have the unit vector. extend the weld distance from the intersection
        |   x = xintersect + l2delxunit * wd
        |   y = yintersect + l2delyunit * wd
        | 
        |   point5 = p[x,y,z,0,-1.570796,0]
        | 
        |   x = xintersect + l2delxunit * rod
        |   y = yintersect + l2delyunit * rod
        | 
        |   point4 = p[x,y,z,0,-1.570796,0]
        | 
        |   #DEFINE APPROACH POINTS
        |   pointintersect = p[xintersect,yintersect,zcoord,0,0,0]
        |   pointapproach1 = p[xintersect+0.1,yintersect+0.1,z,1.570796,0,0]
        |   pointapproach2 = p[point1[0], point1[1]+0.1, point1[2], point1[3], point1[4], point1[5]]
        |   pointreturn1 = p[point5[0]+0.1, point5[1], point5[2], point5[3], point5[4], point5[5]]
        | 
        |   #FIND HEADINGS
        |   #for each heading, find the angle of the line with respect to the pos x axis. then add/subtract 90 degrees because you want to be perpendicular to that
        |   headingvector1 = convert_uv_to_heading(l1delxunit, l1delyunit)
        |   headingvector2 = convert_uv_to_heading(l2delxunit, l2delyunit)
        |   # find halfway heading
        |   heading2 = (headingvector1 + headingvector2)/2
        |   # find headings that the robot should face while traveling, perpendicular to the vectors of the sides of the box
        |   heading1 = headingvector1 + pi/2
        |   heading3 = headingvector2 - pi/2
        | 
        |   #FIND POINT 3
        |   #see if we have to / can find point 3
        |   findpoint3 = True
        |   if roundoverdistance == 0:
        |     findpoint3 = False
        |   end
        |   if findpoint3:
        |     # i need to find the point3 such that the arc from p2 to p3 to p4 is tangent to p1-p2 and p4-p5. making this a smooth path will be good
        |     # the direction of movement is from pointintersect in the direction of heading2
        |     # how much movement though? this will depend on whether it is actually a 90 degree angle or not.
        |     # first, find the perpendicular lines through points 2 and 4
        |     perp2 = find_perpendicular_line(ml1, point2[0], point2[1])
        |     perp4 = find_perpendicular_line(ml2, point4[0], point4[1])
        |     # next, find the intersection of those two lines
        |     perpintersect = find_intersection(perp2[0], perp2[1], perp4[0], perp4[1])
        |     radiusofcircle = distance_between(perpintersect[0], perpintersect[1], 0, point2[0], point2[1], 0)
        |     # find a vector the direction of heading2
        |     uvx = cos(heading2)
        |     uvy = sin(heading2)
        |     # compute point3. pass in negative radius because the direction is into the tank but we want to move from the intersection out to the rounded edge
        |     point3coords = add_vectordistance_to_point(perpintersect[0], perpintersect[1], z, uvx, uvy, 0, -1 * radiusofcircle)
        |     point3 = p[point3coords[0], point3coords[1], point3coords[2], 0, 0, 0]
        |   end
        | 
        |   #APPLY ACTUAL RXRYRZ TO POINTS
        |   # convert the headings to rxryrz and insert those values into the relevant points
        |   rxryrz = convert_heading_to_axang(heading1)
        |   rx = rxryrz[0]
        |   ry = rxryrz[1]
        |   rz = rxryrz[2]
        |   pointapproach1 = p[pointapproach1[0], pointapproach1[1], pointapproach1[2], rx, ry, rz]
        |   pointapproach2 = p[pointapproach2[0], pointapproach2[1], pointapproach2[2], rx, ry, rz]
        |   point1 = p[point1[0], point1[1], point1[2], rx, ry, rz]
        |   point2 = p[point2[0], point2[1], point2[2], rx, ry, rz]
        |   rxryrz = convert_heading_to_axang(heading2)
        |   rx = rxryrz[0]
        |   ry = rxryrz[1]
        |   rz = rxryrz[2]
        |   if findpoint3:
        |     point3 = p[point3[0], point3[1], point3[2], rx, ry, rz]
        |   else:
        |     point3 = point2
        |   end
        |   rxryrz = convert_heading_to_axang(heading3)
        |   rx = rxryrz[0]
        |   ry = rxryrz[1]
        |   rz = rxryrz[2]
        |   point4 = p[point4[0], point4[1], point4[2], rx, ry, rz]
        |   point5 = p[point5[0], point5[1], point5[2], rx, ry, rz]
        |   pointreturn1 = p[pointreturn1[0], pointreturn1[1], pointreturn1[2], rx, ry, rz]
        | 
        |   #find path2 (the part that goes up)
        |   four_vertical_points = find_vertical_points(pointintersect, l1delxunit, l1delyunit, l2delxunit, l2delyunit, zup, wd, heading1, heading3)
        |   path2r1 = four_vertical_points[0]
        |   path2r2 = four_vertical_points[1]
        |   path2l1 = four_vertical_points[2]
        |   path2l2 = four_vertical_points[3]
        | 
        |   #RETURN STRUCT
        |   ret = struct(pointintersect=pointintersect, pointapproach1=pointapproach1, pointapproach2=pointapproach2, point1=point1, point2=point2, point3=point3, point4=point4, point5=point5, pointreturn1=pointreturn1, heading1=heading1, heading2=heading2, heading3=heading3, path2r1=path2r1, path2r2=path2r2, path2l1=path2l1, path2l2=path2l2)
        |   return ret
        | end
        | 
        | # it takes 5 arguments as points
        | # it returns a struct containing: (pointintersect, heading1, heading2, heading3, l1delxunit, l1delyunit, l2delxunit, l2delyunit)
        | def analyze_touchpoints_only(p11, p12, p21, p22, p3):
        |   # FIND THE INTERSECTION
        |   # comment get the z
        |   zcoord=p3[2]
        | 
        |   # get the raw points from the first line
        |   l1p1x=p11[0]
        |   l1p1y=p11[1]
        |   l1p2x=p12[0]
        |   l1p2y=p12[1]
        | 
        |   # equate the first line in 2d space
        |   ml1 = (l1p2y-l1p1y) / (l1p2x-l1p1x)
        | 
        |   # b = y - mx
        |   bl1 = l1p1y - ml1 * l1p1x
        | 
        |   # get the raw points from the second line
        |   l2p1x=p21[0]
        |   l2p1y=p21[1]
        |   l2p2x=p22[0]
        |   l2p2y=p22[1]
        | 
        |   # equate the second line in 2d space
        |   ml2 = (l2p2y-l2p1y) / (l2p2x-l2p1x)
        | 
        |   # b = y - mx
        |   bl2 = l2p1y - ml2 * l2p1x
        | 
        | 
        |   # find the intersection of the two lines
        |   # m1x+b1 = m2x+b2
        |   # m1x - m2x = b2 - b1
        |   # x = (b2-b1) / (m1-m2)
        |   xintersect = (bl2-bl1) / (ml1-ml2)
        |   yintersect = ml1 * xintersect + bl1
        | 
        |   pointintersect = p[xintersect,yintersect,zcoord,0,0,0]
        | 
        |   #FIND THE VECTORS
        |   #define a vector from the intersection to the second point on the first line
        |   l1delxfull = l1p2x - xintersect
        |   l1delyfull = l1p2y - yintersect
        | 
        |   l1delmag = sqrt(l1delxfull*l1delxfull + l1delyfull*l1delyfull)
        | 
        |   l1delxunit = l1delxfull / l1delmag
        |   l1delyunit = l1delyfull / l1delmag
        | 
        |   #define a vector from the intersection to the second point on the second line
        |   l2delxfull = l2p2x - xintersect
        |   l2delyfull = l2p2y - yintersect
        | 
        |   l2delmag = sqrt(l2delxfull*l2delxfull + l2delyfull*l2delyfull)
        | 
        |   l2delxunit = l2delxfull / l2delmag
        |   l2delyunit = l2delyfull / l2delmag
        | 
        |   #FIND HEADINGS
        |   #for each heading, find the angle of the line with respect to the pos x axis. then add/subtract 90 degrees because you want to be perpendicular to that
        |   headingvector1 = convert_uv_to_heading(l1delxunit, l1delyunit)
        |   headingvector2 = convert_uv_to_heading(l2delxunit, l2delyunit)
        |   # find halfway heading
        |   heading2 = (headingvector1 + headingvector2)/2
        |   # find headings that the robot should face while traveling, perpendicular to the vectors of the sides of the box
        |   heading1 = headingvector1 + pi/2
        |   heading3 = headingvector2 - pi/2
        | 
        |   #RETURN STRUCT
        |   ret = struct(pointintersect=pointintersect, heading1=heading1, heading2=heading2, heading3=heading3, l1delxunit=l1delxunit, l1delyunit=l1delyunit, l2delxunit=l2delxunit, l2delyunit=l2delyunit)
        |   return ret
        | end
        | 
        | # given a struct from analyze_touchpoints_only(), calculate the points
        | # for right, for non-extended
        | def calculate_DOtA_points_right(struct1, listleans, chamferover):
        |     # get the stuff from the struct
        |     pointintersect = struct1[0]
        |     heading1 = struct1[1]
        |     heading2 = struct1[2]
        |     heading3 = struct1[3]
        |     l1delxunit = struct1[4]
        |     l1delyunit = struct1[5]
        |     l2delxunit = struct1[6]
        |     l2delyunit = struct1[7]
        | 
        |     # FIND THE POINTS ON THE LINES OF THE FIRST TURN PATH
        |     # find locations 8 inches away from  intersect point
        |     # CONST
        |     welddistance1 = 8 # vertical weld distance
        |     welddistance2 = 6 # first path second leg
        |     welddistance3 = 8 # second path second leg
        |     zup = .375
        |     # inches
        |     wd1 = welddistance1 * 25.4 / 1000
        |     wd2 = welddistance2 * 25.4 / 1000
        |     wd3 = welddistance3 * 25.4 / 1000
        |     zup = zup * 25.4 / 1000
        |     chamferovermm =  chamferover * 25.4 / 1000
        | 
        |     x = pointintersect[0] + l1delxunit * chamferovermm
        |     y = pointintersect[1] + l1delyunit * chamferovermm
        |     z = pointintersect[2] + zup
        | 
        |     #apply actual rxryrz to points
        |     # convert the headings to rxryrz and insert those values into the relevant points
        |     rxryrz = convert_heading_to_axang_preheatdown(heading1)
        |     rx = rxryrz[0]
        |     ry = rxryrz[1]
        |     rz = rxryrz[2]
        | 
        |     point1 = p[x + wd1*listleans[0], y + wd1*listleans[1], z + wd1, rx, ry, rz] # add in the listleans factor to follow the face of the box as we move up
        |     point2 = p[x, y, z, rx, ry, rz]
        | 
        |     # convert the headings to rxryrz and insert those values into the relevant points
        |     rxryrz = convert_heading_to_axang_ccw(heading1)
        |     rx = rxryrz[0]
        |     ry = rxryrz[1]
        |     rz = rxryrz[2]
        | 
        |     point4 = p[x, y, z, rx, ry, rz]
        |     x = x + l1delxunit * wd2
        |     y = y + l1delyunit * wd2
        |     point5 = p[x, y, z, rx, ry, rz]
        | 
        |     # FIND THE POINTS ON THE LINES OF THE SECOND AROUND PATH
        |     roundoverdistance = 0.05
        |     rod = roundoverdistance * 25.4 / 1000
        | 
        |     # now we have the unit vector. extend the weld distance from the intersection
        |     x = pointintersect[0] + l1delxunit * chamferovermm
        |     y = pointintersect[1] + l1delyunit * chamferovermm
        |     # convert the headings to rxryrz and insert those values into the relevant points
        |     rxryrz = convert_heading_to_axang(heading1)
        |     rx = rxryrz[0]
        |     ry = rxryrz[1]
        |     rz = rxryrz[2]
        |     point_1 = p[x, y, z, rx, ry, rz]
        | 
        |     x = pointintersect[0] + l1delxunit * rod
        |     y = pointintersect[1] + l1delyunit * rod
        |     point_2 = p[x, y, z, rx, ry, rz]
        | 
        |     # now we have the unit vector. extend the weld distance from the intersection
        |     x = pointintersect[0] + l2delxunit * wd3
        |     y = pointintersect[1] + l2delyunit * wd3
        |     # convert the headings to rxryrz and insert those values into the relevant points
        |     rxryrz = convert_heading_to_axang(heading3)
        |     rx = rxryrz[0]
        |     ry = rxryrz[1]
        |     rz = rxryrz[2]
        |     point_5 = p[x, y, z, rx, ry, rz]
        | 
        |     x = pointintersect[0] + l2delxunit * rod
        |     y = pointintersect[1] + l2delyunit * rod
        |     point_4 = p[x, y, z, rx, ry, rz]
        | 
        |     #FIND POINT 3
        |     # by calling analyze_touchpoints()
        |     atret = analyze_touchpoints(point_2, point_1, point_4, point_5, pointintersect)
        |     point_3 = atret[5]
        | 
        | 
        |     struct2 = struct(point1=point1, point2=point2, point4=point4, point5=point5, point_1=point_1, point_2=point_2, point_3=point_3, point_4=point_4, point_5=point_5)
        |     return struct2
        | end
        | 
        | # given a struct from analyze_touchpoints_only(), calculate the points
        | # for left, for non-extended
        | def calculate_DOtA_points_left(struct1, listleans, chamferover):
        |     # get the stuff from the struct
        |     pointintersect = struct1[0]
        |     heading1 = struct1[1]
        |     heading2 = struct1[2]
        |     heading3 = struct1[3]
        |     l1delxunit = struct1[4]
        |     l1delyunit = struct1[5]
        |     l2delxunit = struct1[6]
        |     l2delyunit = struct1[7]
        | 
        |     # FIND THE POINTS ON THE LINES OF THE FIRST TURN PATH
        |     # find locations 8 inches away from  intersect point
        |     # CONST
        |     welddistance1 = 8 # vertical weld distance
        |     welddistance2 = 6 # first path second leg
        |     welddistance3 = 8 # second path second leg
        |     zup = .375
        |     # inches
        |     wd1 = welddistance1 * 25.4 / 1000
        |     wd2 = welddistance2 * 25.4 / 1000
        |     wd3 = welddistance3 * 25.4 / 1000
        |     zup = zup * 25.4 / 1000
        |     chamferovermm =  chamferover * 25.4 / 1000
        | 
        |     x = pointintersect[0] + l2delxunit * chamferovermm
        |     y = pointintersect[1] + l2delyunit * chamferovermm
        |     z = pointintersect[2] + zup
        | 
        |     #apply actual rxryrz to points
        |     # convert the headings to rxryrz and insert those values into the relevant points
        |     rxryrz = convert_heading_to_axang_preheatdown(heading3)
        |     rx = rxryrz[0]
        |     ry = rxryrz[1]
        |     rz = rxryrz[2]
        | 
        |     point1 = p[x + wd1*listleans[0], y + wd1*listleans[1], z + wd1, rx, ry, rz]
        |     point2 = p[x, y, z, rx, ry, rz]
        | 
        |     # convert the headings to rxryrz and insert those values into the relevant points
        |     rxryrz = convert_heading_to_axang(heading3)
        |     rx = rxryrz[0]
        |     ry = rxryrz[1]
        |     rz = rxryrz[2]
        | 
        |     point4 = p[x, y, z, rx, ry, rz]
        |     x = x + l2delxunit * wd2
        |     y = y + l2delyunit * wd2
        |     point5 = p[x, y, z, rx, ry, rz]
        | 
        |     # FIND THE POINTS ON THE LINES OF THE SECOND AROUND PATH
        |     roundoverdistance = 0.05
        |     rod = roundoverdistance * 25.4 / 1000
        | 
        |     # now we have the unit vector. extend the weld distance from the intersection
        |     x = pointintersect[0] + l2delxunit * chamferovermm
        |     y = pointintersect[1] + l2delyunit * chamferovermm
        |     # convert the headings to rxryrz and insert those values into the relevant points
        |     rxryrz = convert_heading_to_axang_ccw(heading3)
        |     rx = rxryrz[0]
        |     ry = rxryrz[1]
        |     rz = rxryrz[2]
        |     point_1 = p[x, y, z, rx, ry, rz]
        | 
        |     x = pointintersect[0] + l2delxunit * rod
        |     y = pointintersect[1] + l2delyunit * rod
        |     point_2 = p[x, y, z, rx, ry, rz]
        | 
        |     # now we have the unit vector. extend the weld distance from the intersection
        |     x = pointintersect[0] + l1delxunit * wd3
        |     y = pointintersect[1] + l1delyunit * wd3
        |     # convert the headings to rxryrz and insert those values into the relevant points
        |     rxryrz = convert_heading_to_axang_ccw(heading1)
        |     rx = rxryrz[0]
        |     ry = rxryrz[1]
        |     rz = rxryrz[2]
        |     point_5 = p[x, y, z, rx, ry, rz]
        | 
        |     x = pointintersect[0] + l1delxunit * rod
        |     y = pointintersect[1] + l1delyunit * rod
        |     point_4 = p[x, y, z, rx, ry, rz]
        | 
        |     #FIND POINT 3
        |     # by calling analyze_touchpoints()
        |     atret = analyze_touchpoints(point_2, point_1, point_4, point_5, pointintersect)
        |     point_3 = atret[5]
        |     #point 3 will not have the correct rxryrz though because now the gun needs to be face up.
        |     rxryrz = convert_heading_to_axang_ccw(heading2)
        |     rx = rxryrz[0]
        |     ry = rxryrz[1]
        |     rz = rxryrz[2]
        |     point_3 = p[point_3[0], point_3[1], point_3[2], rx, ry, rz]
        | 
        |     struct2 = struct(point1=point1, point2=point2, point4=point4, point5=point5, point_1=point_1, point_2=point_2, point_3=point_3, point_4=point_4, point_5=point_5)
        |     return struct2
        | end
        | 
        | # given a struct from analyze_touchpoints_only(), calculate the points
        | # for right, for extended
        | def calculate_DOtA_points_right_extended(struct1, listleans, chamferover, chamferup, tcp_pose_top):
        |     # get the stuff from the struct
        |     pointintersect = struct1[0]
        |     heading1 = struct1[1]
        |     heading2 = struct1[2]
        |     heading3 = struct1[3]
        |     l1delxunit = struct1[4]
        |     l1delyunit = struct1[5]
        |     l2delxunit = struct1[6]
        |     l2delyunit = struct1[7]
        | 
        |     # FIND THE POINTS ON THE LINES OF THE FIRST TURN PATH
        |     # find locations 8 inches away from  intersect point
        |     # CONST
        |     # welddistance1 = 8 # vertical weld distance
        |     welddistance2 = 6 # first path second leg
        |     welddistance3 = 8 # second path second leg
        | 
        |     # inches
        |     # wd1 = welddistance1 * 25.4 / 1000
        |     wd2 = welddistance2 * 25.4 / 1000
        |     wd3 = welddistance3 * 25.4 / 1000
        |     zup = chamferup * 25.4 / 1000
        |     chamferovermm =  chamferover * 25.4 / 1000
        | 
        |     # weld distance is the distance that it will weld. this will make it start at the z height that the user specified
        |     wd1 = tcp_pose_top[2] - pointintersect[2] - zup
        | 
        |     x = pointintersect[0] + l1delxunit * chamferovermm
        |     y = pointintersect[1] + l1delyunit * chamferovermm
        |     z = pointintersect[2] + zup
        | 
        |     #apply actual rxryrz to points
        |     # convert the headings to rxryrz and insert those values into the relevant points
        |     rxryrz = convert_heading_to_axang_preheatdown(heading1)
        |     rx = rxryrz[0]
        |     ry = rxryrz[1]
        |     rz = rxryrz[2]
        | 
        |     point1 = p[x + wd1*listleans[0], y + wd1*listleans[1], z + wd1, rx, ry, rz] # add in the listleans factor to follow the face of the box as we move up
        |     point2 = p[x, y, z, rx, ry, rz]
        | 
        |     # convert the headings to rxryrz and insert those values into the relevant points
        |     rxryrz = convert_heading_to_axang_ccw(heading1)
        |     rx = rxryrz[0]
        |     ry = rxryrz[1]
        |     rz = rxryrz[2]
        | 
        |     point4 = p[x, y, z, rx, ry, rz]
        |     x = x + l1delxunit * wd2
        |     y = y + l1delyunit * wd2
        |     point5 = p[x, y, z, rx, ry, rz]
        | 
        |     # FIND THE POINTS ON THE LINES OF THE SECOND AROUND PATH
        |     roundoverdistance = 0.05
        |     rod = roundoverdistance * 25.4 / 1000
        | 
        |     # now we have the unit vector. extend the weld distance from the intersection
        |     x = pointintersect[0] + l1delxunit * chamferovermm
        |     y = pointintersect[1] + l1delyunit * chamferovermm
        |     # convert the headings to rxryrz and insert those values into the relevant points
        |     rxryrz = convert_heading_to_axang(heading1)
        |     rx = rxryrz[0]
        |     ry = rxryrz[1]
        |     rz = rxryrz[2]
        |     point_1 = p[x, y, z, rx, ry, rz]
        | 
        |     x = pointintersect[0] + l1delxunit * rod
        |     y = pointintersect[1] + l1delyunit * rod
        |     point_2 = p[x, y, z, rx, ry, rz]
        | 
        |     # convert the headings to rxryrz and insert those values into the relevant points
        |     rxryrz = convert_heading_to_axang(heading3)
        |     rx = rxryrz[0]
        |     ry = rxryrz[1]
        |     rz = rxryrz[2]
        | 
        |     x = pointintersect[0] + l2delxunit * rod
        |     y = pointintersect[1] + l2delyunit * rod
        |     point_4 = p[x, y, z, rx, ry, rz]
        | 
        |     # now we have the unit vector. extend the weld distance from the intersection
        |     x = pointintersect[0] + l2delxunit * wd3
        |     y = pointintersect[1] + l2delyunit * wd3
        |     point_5 = p[x, y, z, rx, ry, rz]
        | 
        |     #FIND POINT 3
        |     # by calling analyze_touchpoints()
        |     atret = analyze_touchpoints(point_2, point_1, point_4, point_5, pointintersect)
        |     point_3 = atret[5]
        | 
        | 
        |     struct2 = struct(point1=point1, point2=point2, point4=point4, point5=point5, point_1=point_1, point_2=point_2, point_3=point_3, point_4=point_4, point_5=point_5)
        |     return struct2
        | end
        | 
        | # given a struct from analyze_touchpoints_only(), calculate the points
        | # for left, for extended
        | def calculate_DOtA_points_left_extended(struct1, listleans, chamferover, chamferup, tcp_pose_top):
        |     # get the stuff from the struct
        |     pointintersect = struct1[0]
        |     heading1 = struct1[1]
        |     heading2 = struct1[2]
        |     heading3 = struct1[3]
        |     l1delxunit = struct1[4]
        |     l1delyunit = struct1[5]
        |     l2delxunit = struct1[6]
        |     l2delyunit = struct1[7]
        | 
        |     # FIND THE POINTS ON THE LINES OF THE FIRST TURN PATH
        |     # find locations 8 inches away from  intersect point
        |     # CONST
        |     # welddistance1 = 8 # vertical weld distance
        |     welddistance2 = 6 # first path second leg
        |     welddistance3 = 8 # second path second leg
        | 
        |     # inches
        |     # wd1 = welddistance1 * 25.4 / 1000
        |     wd2 = welddistance2 * 25.4 / 1000
        |     wd3 = welddistance3 * 25.4 / 1000
        |     zup = chamferup * 25.4 / 1000
        |     chamferovermm =  chamferover * 25.4 / 1000
        | 
        |     # weld distance is the distance that it will weld. this will make it start at the z height that the user specified
        |     wd1 = tcp_pose_top[2] - pointintersect[2] - zup
        | 
        |     x = pointintersect[0] + l2delxunit * chamferovermm
        |     y = pointintersect[1] + l2delyunit * chamferovermm
        |     z = pointintersect[2] + zup
        | 
        |     #apply actual rxryrz to points
        |     # convert the headings to rxryrz and insert those values into the relevant points
        |     rxryrz = convert_heading_to_axang_preheatdown(heading3)
        |     rx = rxryrz[0]
        |     ry = rxryrz[1]
        |     rz = rxryrz[2]
        | 
        |     point1 = p[x + wd1*listleans[0], y + wd1*listleans[1], z + wd1, rx, ry, rz]
        |     point2 = p[x, y, z, rx, ry, rz]
        | 
        |     # convert the headings to rxryrz and insert those values into the relevant points
        |     rxryrz = convert_heading_to_axang(heading3)
        |     rx = rxryrz[0]
        |     ry = rxryrz[1]
        |     rz = rxryrz[2]
        | 
        |     point4 = p[x, y, z, rx, ry, rz]
        |     x = x + l2delxunit * wd2
        |     y = y + l2delyunit * wd2
        |     point5 = p[x, y, z, rx, ry, rz]
        | 
        |     # FIND THE POINTS ON THE LINES OF THE SECOND AROUND PATH
        |     roundoverdistance = 0.05
        |     rod = roundoverdistance * 25.4 / 1000
        | 
        |     # now we have the unit vector. extend the weld distance from the intersection
        |     x = pointintersect[0] + l2delxunit * chamferovermm
        |     y = pointintersect[1] + l2delyunit * chamferovermm
        |     # convert the headings to rxryrz and insert those values into the relevant points
        |     rxryrz = convert_heading_to_axang_ccw(heading3)
        |     rx = rxryrz[0]
        |     ry = rxryrz[1]
        |     rz = rxryrz[2]
        |     point_1 = p[x, y, z, rx, ry, rz]
        | 
        |     x = pointintersect[0] + l2delxunit * rod
        |     y = pointintersect[1] + l2delyunit * rod
        |     point_2 = p[x, y, z, rx, ry, rz]
        | 
        |     # convert the headings to rxryrz and insert those values into the relevant points
        |     rxryrz = convert_heading_to_axang_ccw(heading1)
        |     rx = rxryrz[0]
        |     ry = rxryrz[1]
        |     rz = rxryrz[2]
        | 
        |     x = pointintersect[0] + l1delxunit * rod
        |     y = pointintersect[1] + l1delyunit * rod
        |     point_4 = p[x, y, z, rx, ry, rz]
        | 
        |     # now we have the unit vector. extend the weld distance from the intersection
        |     x = pointintersect[0] + l1delxunit * wd3
        |     y = pointintersect[1] + l1delyunit * wd3
        |     point_5 = p[x, y, z, rx, ry, rz]
        | 
        |     #FIND POINT 3
        |     # by calling analyze_touchpoints()
        |     atret = analyze_touchpoints(point_2, point_1, point_4, point_5, pointintersect)
        |     point_3 = atret[5]
        |     #point 3 will not have the correct rxryrz though because now the gun needs to be face up
        |     rxryrz = convert_heading_to_axang_ccw(heading2)
        |     rx = rxryrz[0]
        |     ry = rxryrz[1]
        |     rz = rxryrz[2]
        |     point_3 = p[point_3[0], point_3[1], point_3[2], rx, ry, rz]
        | 
        |     struct2 = struct(point1=point1, point2=point2, point4=point4, point5=point5, point_1=point_1, point_2=point_2, point_3=point_3, point_4=point_4, point_5=point_5)
        |     return struct2
        | end
        | 
        | # this function analyzes the vertical points
        | # calculates the slope of the edge in question
        | # specifically, for each inch up in the z direction, what is the change in x and change in y direction
        | # returns a list of [nx, ny]
        | def analyze_vertical_touchpoints(p11, p12, p13, p21, p22, p23, p3):
        |     # first, find the equations of the planes from the 6 points
        |     plane1 = findplane(p11, p12, p13)
        |     plane2 = findplane(p21, p22, p23)
        |     # Find the Direction Vector of the Line: The direction vector d of the line of intersection can be found by taking the cross product of the normal vectors of each plane (a, b, and c)
        |     nx = plane1[1]*plane2[2] - plane1[2]*plane2[1]
        |     ny = plane1[2]*plane2[0] - plane1[0]*plane2[2]
        |     nz = plane1[0]*plane2[1] - plane1[1]*plane2[0]
        |     # normalize the vector so the z length is 1
        |     multiplier = 1 / nz
        |     nx = nx * multiplier
        |     ny = ny * multiplier
        |     nz = nz * multiplier # should become equal to 1
        |     ret = [nx, ny]
        |     return ret
        | end
        | 
        | # given 3 points, this finds the plane and its equation
        | # rereturns ax + by + cz + d = 0 in a list of [a, b, c, d]
        | def findplane(p11, p12, p13):
        |     # extract coordinates
        |     x1 = p11[0]
        |     y1 = p11[1]
        |     z1 = p11[2]
        |     x2 = p12[0]
        |     y2 = p12[1]
        |     z2 = p12[2]
        |     x3 = p13[0]
        |     y3 = p13[1]
        |     z3 = p13[2]
        |     # create vectors from the points
        |     v1x = x2-x1
        |     v1y = y2-y1
        |     v1z = z2-z1
        |     v2x = x3-x1
        |     v2y = y3-y1
        |     v2z = z3-z1
        |     #calculate the normal vector using the cross product
        |     nx = v1y*v2z - v1z*v2y # i component
        |     ny = v1z*v2x - v1x*v2z # j component
        |     nz = v1x*v2y - v1y*v2x # k component
        |     # calculate d in the plane equation
        |     d = -1 * (nx*x1 + ny*y1 + nz*z1)
        |     ret = [nx, ny, nz, d]
        |     return ret
        | end
        | 
        | # given a heading, (ccw from +x axis), find the mx+b slope
        | # fails if exactly vertical
        | def get_slope_from_heading(heading):
        |     return tan(heading)
        | end
        | 
        | 
        | 
        | # this function finds the points (and rxryrz) of the 2 points (start and end) of vertical weld section
        | def find_vertical_points(pointintersect, l1delxunit, l1delyunit, l2delxunit, l2delyunit, offset, wd, heading1, heading3):
        | 
        |   # find right side stuff
        |   # find the point in 3d space that is .375 up and .375 over
        |   x = pointintersect[0] + l1delxunit * offset
        |   y = pointintersect[1] + l1delyunit * offset
        |   z = pointintersect[2] + offset
        |   # find rxryrz
        |   rxryrz = convert_heading_to_axang_preheatup(heading1)
        |   rx = rxryrz[0]
        |   ry = rxryrz[1]
        |   rz = rxryrz[2]
        |   path2r1 = p[x, y, z, rx, ry, rz]
        |   path2r2 = p[x, y, z + wd, rx, ry, rz]
        | 
        |   # find left side
        |   # find the point in 3d space that is .375 up and .375 over
        |   x = pointintersect[0] + l2delxunit * offset
        |   y = pointintersect[1] + l2delyunit * offset
        |   z = pointintersect[2] + offset
        |   # find rxryrz
        |   rxryrz = convert_heading_to_axang_preheatup(heading3)
        |   rx = rxryrz[0]
        |   ry = rxryrz[1]
        |   rz = rxryrz[2]
        |   path2l1 = p[x, y, z, rx, ry, rz]
        |   path2l2 = p[x, y, z + wd, rx, ry, rz]
        | 
        |   ret = struct(path2r1=path2r1, path2r2=path2r2, path2l1=path2l1, path2l2=path2l2)
        |   return ret
        | end
        | 
        | # this function converts a unit vector to its heading angle ccw from x+ axis
        | # takes uvx and uvy
        | # returns heading in radians
        | def convert_uv_to_heading(uvx, uvy):
        |   baseang = atan(uvy/uvx)
        |   if uvx < 0:
        |     ang = baseang + pi
        |   elif uvy < 0:
        |     ang = baseang + pi * 2
        |   else:
        |     ang = baseang
        |   end
        |   return ang
        | end
        | 
        | # this function finds the equation of a line, perpendicular to a given line, and going through a given point
        | # takes 3 arguments: m (the original line's slope), x (point's x coord), y (point's y coord). the b of the original line is not needed
        | # returns a list of [m,b] (the slope and intercept of the new line)
        | def find_perpendicular_line(origm, x, y):
        |   m = (1/origm) * -1
        |   b = y - m*x
        |   ret = [m, b]
        |   return ret
        | end
        | 
        | # this function finds the intersection point between two lines in the xy plane
        | # takes 4 arguments: m1, b1, m2, b2
        | # returns a list of [x,y] (the point of intersection)
        | def find_intersection(m1, b1, m2, b2):
        |   # m1x+b1 = m2x+b2
        |   # m1x - m2x = b2 - b1
        |   # x = (b2-b1) / (m1-m2)
        |   x = (b2-b1) / (m1-m2)
        |   y = m1 * x + b1
        |   ret = [x, y]
        |   return ret
        | end
        | 
        | # this function finds the distance between 2 points in 3d space
        | # it takes 6 arguments: x1, y1, z1, x2, y2, z2
        | # it returns a distance
        | def distance_between(x1, y1, z1, x2, y2, z2):
        |   distsquared = (x2-x1)*(x2-x1)+(y2-y1)*(y2-y1)+(z2-z1)*(z2-z1)
        |   dist = sqrt(distsquared)
        |   return dist
        | end
        | 
        | # this function takes a point, a unit vector, and a distance, and adds the distance to the point in the direction of the unit vector (3d space)
        | # it returns a point as a list of coordinates
        | def add_vectordistance_to_point(xi, yi, zi, uvx, uvy, uvz, delta):
        |   xf = xi + uvx * delta
        |   yf = yi + uvy * delta
        |   zf = zi + uvz * delta
        |   ret = [xf, yf, zf]
        |   return ret
        | end
        | 
        | # this function converts a heading (ccw radians from the positive x axis) into rxryrz to be put into a point p[]
        | # this will point the gun in this heading with the bottom side of the gun facing up.
        | # the values used in this program were calculated by doing rotation matrix math in the file on WI-CALVINB10 C. Documents. Theory for converting rotations into axis angle representations
        | def convert_heading_to_axang(heading):
        |  axisxraw = -1 * sin(heading)
        |  axisyraw = cos(heading) + 1
        |  axiszraw = sin(heading)
        | 
        |  magnitude = sqrt(axisxraw*axisxraw + axisyraw*axisyraw + axiszraw*axiszraw)
        | 
        |  axisxunit = axisxraw / magnitude
        |  axisyunit = axisyraw / magnitude
        |  axiszunit = axiszraw / magnitude
        | 
        |  angle = acos( (cos(heading) - 1) / 2 )
        | 
        |  rxout = axisxunit * angle
        |  ryout = axisyunit * angle
        |  rzout = axiszunit * angle
        | 
        |  return [rxout, ryout, rzout]
        | end
        | 
        | # this function converts a heading (ccw radians from the positive x axis) into rxryrz to be put into a point p[]
        | # this will point the gun in this heading with the preheat side of the gun tip facing up. Used for welding in a vertical path.
        | # the values used in this program were calculated by doing rotation matrix math in the file on WI-CALVINB10 C. Documents. Theory for converting rotations into axis angle representations
        | def convert_heading_to_axang_preheatup(heading):
        |  axisxraw = -sin(heading) + 1
        |  axisyraw = cos(heading)
        |  axiszraw = cos(heading)
        | 
        |  magnitude = sqrt(axisxraw*axisxraw + axisyraw*axisyraw + axiszraw*axiszraw)
        | 
        |  axisxunit = axisxraw / magnitude
        |  axisyunit = axisyraw / magnitude
        |  axiszunit = axiszraw / magnitude
        | 
        |  angle = acos( (-sin(heading) - 1) / 2 )
        | 
        |  rxout = axisxunit * angle
        |  ryout = axisyunit * angle
        |  rzout = axiszunit * angle
        | 
        |  return [rxout, ryout, rzout]
        | end
        | 
        | # this function converts a heading (ccw radians from the positive x axis) into rxryrz to be put into a point p[]
        | # this will point the gun in this heading with the preheat side of the gun tip facing down. Used for welding in a vertical path downwards.
        | # the values used in this program were calculated by doing rotation matrix math in the file on WI-CALVINB10 C. Documents. Theory for converting rotations into axis angle representations
        | def convert_heading_to_axang_preheatdown(heading):
        |  axisxraw = -sin(heading) - 1
        |  axisyraw = cos(heading)
        |  axiszraw = -cos(heading)
        | 
        |  magnitude = sqrt(axisxraw*axisxraw + axisyraw*axisyraw + axiszraw*axiszraw)
        | 
        |  axisxunit = axisxraw / magnitude
        |  axisyunit = axisyraw / magnitude
        |  axiszunit = axiszraw / magnitude
        | 
        |  angle = acos( (sin(heading) - 1) / 2 )
        | 
        |  rxout = axisxunit * angle
        |  ryout = axisyunit * angle
        |  rzout = axiszunit * angle
        | 
        |  return [rxout, ryout, rzout]
        | end
        | 
        | # this function converts a heading (ccw radians from the positive x axis) into rxryrz to be put into a point p[]
        | # this will point the gun in this heading with the preheat side of the gun tip facing right. Used for welding counterclockwise around the box.
        | # the values used in this program were calculated by doing rotation matrix math in the file on WI-CALVINB10 C. Documents. Theory for converting rotations into axis angle representations
        | def convert_heading_to_axang_ccw(heading):
        |  axisxraw = -sin(heading)
        |  axisyraw = cos(heading) - 1
        |  axiszraw = -sin(heading)
        | 
        |  magnitude = sqrt(axisxraw*axisxraw + axisyraw*axisyraw + axiszraw*axiszraw)
        | 
        |  axisxunit = axisxraw / magnitude
        |  axisyunit = axisyraw / magnitude
        |  axiszunit = axiszraw / magnitude
        | 
        |  angle = acos( (-cos(heading) - 1) / 2 )
        | 
        |  rxout = axisxunit * angle
        |  ryout = axisyunit * angle
        |  rzout = axiszunit * angle
        | 
        |  return [rxout, ryout, rzout]
        | end
        | 
        | # this function takes two rotation matrices, and multiplies them together, returning one matrix.
        | # all matrices are in the form of a list.
        | # all matrix values have constant values (no variables)
        | def multiply_matrix(matrix1, matrix2):
        |     # retrieve values
        |     a11 = matrix1[0]
        |     a12 = matrix1[1]
        |     a13 = matrix1[2]
        |     a21 = matrix1[3]
        |     a22 = matrix1[4]
        |     a23 = matrix1[5]
        |     a31 = matrix1[6]
        |     a32 = matrix1[7]
        |     a33 = matrix1[8]
        |     b11 = matrix2[0]
        |     b12 = matrix2[1]
        |     b13 = matrix2[2]
        |     b21 = matrix2[3]
        |     b22 = matrix2[4]
        |     b23 = matrix2[5]
        |     b31 = matrix2[6]
        |     b32 = matrix2[7]
        |     b33 = matrix2[8]
        |     #calculate c values
        |     c11 = a11*b11 + a12*b21 + a13*b31
        |     c12 = a11*b12 + a12*b22 + a13*b32
        |     c13 = a11*b13 + a12*b23 + a13*b33
        |     c21 = a21*b11 + a22*b21 + a23*b31
        |     c22 = a21*b12 + a22*b22 + a23*b32
        |     c23 = a21*b13 + a22*b23 + a23*b33
        |     c31 = a31*b11 + a32*b21 + a33*b31
        |     c32 = a31*b12 + a32*b22 + a33*b32
        |     c33 = a31*b13 + a32*b23 + a33*b33
        |     # return resulting matrix
        |     ret = [c11, c12, c13, c21, c22, c23, c31, c32, c33]
        |     return ret
        | end
        | 
        | # this function converts a matrix to axis angle representations
        | # this matrix is usually a resulting matrix (result of matrix multiplication) in normal use, given as a list
        | # returns a list of [rx,ry,rz]
        | def convert_matrix_to_axang(matrix1):
        |     # retrieve values
        |     a11 = matrix1[0]
        |     a12 = matrix1[1]
        |     a13 = matrix1[2]
        |     a21 = matrix1[3]
        |     a22 = matrix1[4]
        |     a23 = matrix1[5]
        |     a31 = matrix1[6]
        |     a32 = matrix1[7]
        |     a33 = matrix1[8]
        | 
        |     # First Half: find the angle
        |     # find the trace
        |     # using the formula: trace = a11 + a22 + a33
        |     trace = a11 + a22 + a33
        |     # find the angle using the formula: trace(matrix) = 1 + 2 cos(angle)
        |     angle = acos((trace - 1.0)/2.0)
        | 
        |     # Second Half: calculate the rotation axis
        |     axisxraw = a32 - a23
        |     axisyraw = a13 - a31
        |     axiszraw = a21 - a12
        |     # normalize axis
        |     magnitude = sqrt(axisxraw*axisxraw + axisyraw*axisyraw + axiszraw*axiszraw)
        |     axisxunit = axisxraw / magnitude
        |     axisyunit = axisyraw / magnitude
        |     axiszunit = axiszraw / magnitude
        | 
        |     # combine axis and angle into rxryrz representation
        |     rxout = axisxunit * angle
        |     ryout = axisyunit * angle
        |     rzout = axiszunit * angle
        |     return [rxout, ryout, rzout]
        | end
        | 
        | # this function takes a rotation and calculates the corresponding rotation matrix
        | # input is (axis, direction, angle in radians)
        | # example is ("x", 1, pi/6) = a 30 degree turn around the x axis in the positive direction (right hand rule)
        | # returns a matrix (a list of 9 values)
        | def get_rotation_matrix_from_description(axis, direction, angle):
        |     # get the angle
        |     a = angle * direction
        |     # get the axis
        |     if axis == "x" or axis == "X":
        |         matrix = [1, 0, 0, 0, cos(a), -1 * sin(a), 0, sin(a), cos(a)]
        |         return matrix
        |     end
        |     if axis == "y" or axis == "Y":
        |         matrix = [cos(a), 0, sin(a), 0, 1, 0, -1*sin(a), 0, cos(a)]
        |         return matrix
        |     end
        |     if axis == "z" or axis == "Z":
        |         matrix = [cos(a), -1*sin(a), 0, sin(a), cos(a), 0, 0, 0, 1]
        |         return matrix
        |     end
        |     # bad
        |     popuptext = "Error in get_rotation_matrix_from_description. "
        |     # infinite loop
        |     while 1==1:
        |       popup(popuptext, title="Code Error",blocking=True)
        |     end
        | end
        | 
        | # this function is for getting the points along the path of the corner homing 45
        | # point0 is the point where they touched
        | def get_corner_homing_45_pathpoints(point0, pointtop = p[0,0,0,0,0,0]):
        |   p0x = point0[0]
        |   p0y = point0[1]
        |   p0z = point0[2]
        |   p0rx = point0[3]
        |   p0ry = point0[4]
        |   p0rz = point0[5]
        | 
        |   #constants
        |   #distances of how far away from point the touchpoints are
        |   d0 = 0.10 # how far from the box to retreat and approach
        |   d1 = 0.03 # first distance from init point
        |   d2 = 0.15 # second distance from init point
        |   d3 = 0.125 #vertical distance from first point
        |   sqrt2 = 0.707106781 # 1/sqrt(2) , the inverse of the sqrt(2)
        | 
        |   ph1 = p[p0x + d0, p0y, p0z + d1, p0rx, p0ry, p0rz] #approach point for turn
        | 
        |   ph2 = p[p0x+d0-d0*0.5-sqrt2*d1, p0y+d0*0.5+sqrt2*d1, p0z+d1, 1.446, -0.8, -0.733]
        |   ph3 = p[p0x+d0-d0*0.5-sqrt2*d2, p0y+d0*0.5+sqrt2*d2, p0z+d1, 1.446, -0.8, -0.733]
        |   ph4 = p[p0x+d0-d0*0.5-sqrt2*d1, p0y-d0*0.5-sqrt2*d1, p0z+d1, 0.626, -1.993, -1.813]
        |   ph5 = p[p0x+d0-d0*0.5-sqrt2*d2, p0y-d0*0.5-sqrt2*d2, p0z+d1, 0.626, -1.993, -1.813]
        | 
        |   # go back to ph1
        |   ph6 = p[p0x + d0, p0y, p0z -0.05, 0, 0, 0] # approach point for under turn
        |   # moveL from ph1 to ph6
        |   ph7 = p[p0x-d1, p0y, p0z-0.05, 0, 0, 0]
        | 
        |   # add the vertical touch points
        |   if pointtop[2] == 0:
        |     ph2up = p[ph2[0], ph2[1], ph2[2]+d3, ph2[3], ph2[4], ph2[5]]
        |     ph4up = p[ph4[0], ph4[1], ph4[2]+d3, ph4[3], ph4[4], ph4[5]]
        |   elif pointtop[2] > p0z + 0.914: # 0.914m = 36 inches
        |     ph2up = p[ph2[0], ph2[1], p0z + 0.914, ph2[3], ph2[4], ph2[5]]
        |     ph4up = p[ph4[0], ph4[1], p0z + 0.914, ph4[3], ph4[4], ph4[5]]
        |   else:
        |     ph2up = p[ph2[0], ph2[1], pointtop[2], ph2[3], ph2[4], ph2[5]]
        |     ph4up = p[ph4[0], ph4[1], pointtop[2], ph4[3], ph4[4], ph4[5]]
        |   end
        |   ret = struct(ph1=ph1, ph2=ph2, ph3=ph3, ph4=ph4, ph5=ph5, ph6=ph6, ph7=ph7, ph2up=ph2up, ph4up=ph4up)
        |   is_robot_at_reachable_spot(point0, ret)
        |   return ret
        | end
        | 
        | # this function checks whether the touchpoints are reachable AKA is the robot positioned in the right spot
        | # if everything looks good, it continues.
        | # if it detects a problem, it infinite loops a popup
        | def is_robot_at_reachable_spot(point0, struct_touchpoints):
        |   # first, check whether the corner is too low to the ground that the bottom homing will hit the ground (z < -400)
        |   lc_height = get_lift_column_height_condensed()
        |   # total height = zeroed lift column height (41.25 inches) (1.04775 m) plus lift column height plus robot relative height
        |   totalheight = 1.04775 + lc_height + point0[2]
        |   if totalheight < 1.04775 - 0.400:
        |     # bad
        |     popuptext = "Tank Corner is too low to the ground. Collisions will occur. Stop Program and raise tank. "
        |     # infinite loop
        |     while 1==1:
        |       popup(popuptext, title="Robot Positioning Warning",blocking=True)
        |     end
        |   end
        | 
        | 
        | 
        |   # next, check whether the touchpoints are reachable
        |   allvalid = check_structofpoints_validity(struct_touchpoints)
        |   if not allvalid:
        | 
        |     # then unreachable
        |     # generate message
        |     listproblems = ""
        |     listnames = ["ph1", "ph2", "ph3", "ph4", "ph5", "ph6", "ph7", "ph2up", "ph4up"]
        |     i = 0
        |     structlength = 9
        |     while i < structlength:
        |       curr = struct_touchpoints[i]
        |       valid = get_inverse_kin_has_solution(curr)
        |       if not valid:
        |         listproblems = listproblems + listnames[i]
        |       end
        |       i = i + 1
        |     end
        |     # display
        |     popuptext = "Robot is too far from tank corner. Cannot reach some necessary positions. Stop Program and move robot closer. " + listproblems
        |     # infinite loop
        |     while 1==1:
        |       popup(popuptext, title="Robot Positioning Warning",blocking=True)
        |     end
        |   end
        | 
        | end
        | 
        | # this function takes a struct of points as an argument, and checks whether every point in the list is reachable using get_inverse_kin_has_solution()
        | # this function does NOT check for weird twists or joint limits
        | # inputstruct must contain only points
        | # it returns true if all points are valid. it returns false if any points are valid
        | # a list of length 0 indicates that all points are valid
        | def check_structofpoints_validity(inputstruct):
        |   # next, check whether the touchpoints are reachable
        |   structlength = length(inputstruct)
        |   i = 0
        |   allvalid = True
        |   while i < structlength:
        |     curr = inputstruct[i]
        |     valid = get_inverse_kin_has_solution(curr)
        |     if not valid:
        |       return False
        |     end
        |     i = i + 1
        |   end
        |   return True
        | end
        | 
        | # checks the validity of all points during a left weld
        | # takes 2 arguments: struct1 (struct1[0] has to contain pointintersect) and struct2 (contains all the points (9) of the weld path)
        | def check_validity_left(struct1, struct2):
        |   #first, check whether robot is too close
        |   pointintersect = struct1[0]
        |   # next, check if the corner is too close to the robot to do a left around weld (complex but approximately X > -1300)
        |   # if y < 0, then x < -1300. if y < 480, then y > (1300+x)*8. if y > 480, then y > (1235+x)*4 + 500
        |   toocloseleftweld = False
        |   if pointintersect[1] < 0:
        |     if pointintersect[0] > -1.300:
        |       toocloseleftweld = True
        |     end
        |   elif pointintersect[1] < 0.480:
        |     if pointintersect[1] < (1.300 + pointintersect[0])*8:
        |       toocloseleftweld = True
        |     end
        |   else:
        |     if pointintersect[1] < (1.235 + pointintersect[0])*4 + 0.500:
        |       toocloseleftweld = True
        |     end
        |   end
        |   if toocloseleftweld:
        |     # bad
        |     popuptext = "Robot is too close to tank corner. Collisions may occur. Stop Program and move robot farther. "
        |     # infinite loop
        |     while 1==1:
        |       popup(popuptext, title="Robot Positioning Warning",blocking=True)
        |     end
        |   end
        | 
        |   #next, check whether all the points in the weldpath are valid
        |   structlength = 9
        |   i = 0
        |   allvalid = True
        |   listproblems = ""
        |   listnames = ["point1", "point2", "point4", "point5", "point_1", "point_2", "point_3", "point_4", "point_5"]
        |   while i < structlength:
        |     curr = struct2[i]
        |     valid = get_inverse_kin_has_solution(curr)
        |     if not valid:
        |       allvalid = False
        |       listproblems = listproblems + listnames[i]
        |     end
        |     i = i + 1
        |   end
        | 
        |   if not allvalid:
        |     # display
        |     popuptext = "Robot is too far from tank corner. Cannot reach some necessary positions. Stop Program and move robot closer. " + listproblems
        |     # infinite loop
        |     while 1==1:
        |       popup(popuptext, title="Robot Positioning Warning",blocking=True)
        |     end
        |   end
        | 
        |   # check whether the path involves weird turns or joint limits. currently just checks the first position
        |   p_prev = [-0.021118, -1.26292, 2.43578, 5.07088, -2.29912, 1.53362] #last point of left weld prerotate
        |   joints_1 = get_inverse_kin(struct2[0], p_prev) # struct2[0] is point1
        |   allGood = True
        |   i = 0
        |   structlength = 6
        |   while i < structlength:
        |     joint_curr = joints_1[i]
        |     # check for anything that exceeds joint limits
        |     degreesmax = 360 * pi / 180
        |     if joint_curr > degreesmax or joint_curr < degreesmax * -1:
        |       allGood = False
        |     end
        |     # check for anything that is significantly different than the aligned approach. could indicate a twist is needed. we dont want that
        |     maxdifference = 150 * pi / 180
        |     difference = joint_curr - p_prev[i]
        |     if difference > maxdifference or difference * -1 > maxdifference:
        |       allGood = False
        |     end
        |     i = i + 1
        |   end
        | 
        |   if not allGood:
        |     # call lift column extend function
        |     struct2 = floor_corner_lift_column_extend_left(struct2)
        | 
        |   end
        | 
        |   # return struct2 back
        |   return struct2
        | end
        | 
        | # checks the validity of all points during a right weld
        | def check_validity_right(struct1, struct2):
        |   # first, check whether the right pivot will bonk itself
        |   pointintersect = struct1[0]
        |   heading1 = struct1[1] # this is the direction that the welder will face when doing the right side of the box
        | 
        |   #first, check whether the heading is just too far offset
        |   # more than 15 degrees off of 45 is too much
        |   # normal heading is 216 degrees
        |   #201 degrees to 231 degrees
        |   heading1degrees = heading1 * 180 / pi
        |   if heading1degrees < 201 or heading1degrees > 231 :
        |     # then out of range
        |     popuptext = "Robot is not aligned at a 45 degree angle of corner (15 degree leeway). Collisions may occur. Stop Program and align robot. heading1degrees=" + str_cat("",heading1degrees)
        |     # infinite loop
        |     while 1==1:
        |       popup(popuptext, title="Robot Positioning Warning",blocking=True)
        |     end
        |   end
        | 
        |   #TODO: add the checks for whether x is too close, given the heading
        |   # add checks for whether x is too close, given the heading
        |   # different equations for whether heading offset > 5 degrees or less (inc. negative)
        |   headingoffset = heading1degrees - 216
        |   if headingoffset < 5:
        |     # then calculate a and b
        |     a = 0.4584 + -0.02369 * headingoffset
        |     b = (-1151.4 + 13.83 * headingoffset) / 1000
        |     # check whether x > a*y+b
        |     if pointintersect[0] > a * pointintersect[1] + b:
        |       # bad
        |       popuptext = "Robot is too close to tank corner or not at the right angle. Collisions may occur. Stop Program and align robot. "
        |       # infinite loop
        |       while 1==1:
        |         popup(popuptext, title="Robot Positioning Warning",blocking=True)
        |       end
        |     end
        |   else:
        |     # headingoffset > 5 degrees
        |     if pointintersect[1] < 0:
        |       if pointintersect[0] > -1150.0 / 1000.0:
        |         #bad
        |         popuptext = "Robot is too close to tank corner. Collisions may occur. Stop Program and align robot. "
        |         # infinite loop
        |         while 1==1:
        |           popup(popuptext, title="Robot Positioning Warning",blocking=True)
        |         end
        |       end
        |     else:
        |       # if x > .7736 y - 1101.9 then bad
        |       if pointintersect[0] > 0.7736 * pointintersect[1] - 1101.9 / 1000:
        |         popuptext = "Robot is too close to tank corner. Collisions may occur. Stop Program and align robot. "
        |         # infinite loop
        |         while 1==1:
        |           popup(popuptext, title="Robot Positioning Warning",blocking=True)
        |         end
        |       end
        |     end
        |   end
        | 
        |   #next, check whether all the points in the weldpath are valid
        |   structlength = 9
        |   i = 0
        |   allvalid = True
        |   listproblems = ""
        |   listnames = ["point1", "point2", "point4", "point5", "point_1", "point_2", "point_3", "point_4", "point_5"]
        |   while i < structlength:
        |     curr = struct2[i]
        |     valid = get_inverse_kin_has_solution(curr)
        |     if not valid:
        |       allvalid = False
        |       listproblems = listproblems + listnames[i]
        |     end
        |     i = i + 1
        |   end
        | 
        |   if not allvalid:
        |     # display
        |     popuptext = "Robot is too far from tank corner. Cannot reach some necessary positions. Stop Program and move robot closer. " + listproblems
        |     # infinite loop
        |     while 1==1:
        |       popup(popuptext, title="Robot Positioning Warning",blocking=True)
        |     end
        |   end
        | 
        |   # check whether the path involves weird turns or joint limits. currently just checks the first position
        |   p_prev = [-1.13307, -1.48911, 2.84785, 4.92357, -4.89059, 1.57184] #last point of right weld prerotate
        |   joints_1 = get_inverse_kin(struct2[0], p_prev) # struct2[0] is point1
        |   allGood = True
        |   i = 0
        |   structlength = 6
        |   while i < structlength:
        |     joint_curr = joints_1[i]
        |     # check for anything that exceeds joint limits
        |     degreesmax = 360 * pi / 180
        |     if joint_curr > degreesmax or joint_curr < degreesmax * -1:
        |       allGood = False
        |     end
        |     # check for anything that is significantly different than the aligned approach. could indicate a twist is needed. we dont want that
        |     maxdifference = 150 * pi / 180
        |     difference = joint_curr - p_prev[i]
        |     if difference > maxdifference or difference * -1 > maxdifference:
        |       allGood = False
        |     end
        |     i = i + 1
        |   end
        | 
        |   if not allGood:
        |     struct2 = floor_corner_lift_column_extend_right(struct2)
        |   end
        | 
        |   # return struct2 back
        |   return struct2
        | end
        | 
        | def floor_corner_lift_column_extend_right(struct2):
        |   # we know that p1 cannot be accessed without a twist
        |   # calculate the height needed to get to p1
        |   liftcolumnincrement = 2.0 # mm
        |   enoughHeightAdded = False
        |   liftColumnHeightTest = 0
